LIN {X 0,Y 385.568,Z 378.768,A -85,B 0,C 180,E1 18476.822,E2 18476.822} C_VEL
LIN {X 0,Y 385.563,Z 378.767,A -85,B 0,C 180,E1 18472.892,E2 18472.892} C_VEL
LIN {X 0,Y 385.562,Z 378.769,A -85,B 0,C 180,E1 18468.915,E2 18468.915} C_VEL
LIN {X 0,Y 385.555,Z 378.77,A -85,B 0,C 180,E1 18465.03,E2 18465.03} C_VEL
LIN {X 0,Y 385.557,Z 378.769,A -85,B 0,C 180,E1 18461.064,E2 18461.064} C_VEL
LIN {X 0,Y 385.556,Z 378.767,A -85,B 0,C 180,E1 18457.001,E2 18457.001} C_VEL
LIN {X 0,Y 385.568,Z 378.766,A -85,B 0,C 180,E1 18454.536,E2 18454.536} C_VEL
LIN {X 0,Y 384.625,Z 378.889,A -85,B 0,C 180,E1 18453.392,E2 18453.392} C_VEL
LIN {X 0,Y 380.036,Z 379.462,A -85,B 0,C 180,E1 18451.232,E2 18451.232} C_VEL
LIN {X 0,Y 377.78,Z 379.738,A -85,B 0,C 180,E1 18449.743,E2 18449.743} C_VEL
LIN {X 0,Y 377.623,Z 379.753,A -85,B 0,C 180,E1 18449.318,E2 18449.318} C_VEL
LIN {X 0,Y 377.624,Z 379.757,A -85,B 0,C 180,E1 18445.292,E2 18445.292} C_VEL
LIN {X 0,Y 377.628,Z 379.756,A -85,B 0,C 180,E1 18441.32,E2 18441.32} C_VEL
LIN {X 0,Y 377.629,Z 379.756,A -85,B 0,C 180,E1 18437.305,E2 18437.305} C_VEL
LIN {X 0,Y 377.638,Z 379.756,A -85,B 0,C 180,E1 18433.384,E2 18433.384} C_VEL
LIN {X 0,Y 377.639,Z 379.756,A -85,B 0,C 180,E1 18429.382,E2 18429.382} C_VEL
LIN {X 0,Y 377.647,Z 379.757,A -85,B 0,C 180,E1 18425.438,E2 18425.438} C_VEL
LIN {X 0,Y 377.646,Z 379.757,A -85,B 0,C 180,E1 18421.366,E2 18421.366} C_VEL
LIN {X 0,Y 377.655,Z 379.76,A -85,B 0,C 180,E1 18417.489,E2 18417.489} C_VEL
LIN {X 0,Y 377.649,Z 379.762,A -85,B 0,C 180,E1 18413.343,E2 18413.343} C_VEL
LIN {X 0,Y 377.656,Z 379.759,A -85,B 0,C 180,E1 18409.36,E2 18409.36} C_VEL
LIN {X 0,Y 377.646,Z 379.758,A -85,B 0,C 180,E1 18405.23,E2 18405.23} C_VEL
LIN {X 0,Y 377.654,Z 379.759,A -85,B 0,C 180,E1 18401.242,E2 18401.242} C_VEL
LIN {X 0,Y 377.626,Z 379.853,A -85,B 0,C 180,E1 18398.318,E2 18398.318} C_VEL
LIN {X 0,Y 382.854,Z 398.245,A -85,B 0,C 180,E1 18394.648,E2 18394.648} C_VEL
LIN {X 0,Y 387.617,Z 416.474,A -85,B 0,C 180,E1 18391.231,E2 18391.231} C_VEL
LIN {X 0,Y 387.818,Z 419.084,A -85,B 0,C 180,E1 18390.79,E2 18390.79} C_VEL
LIN {X 0,Y 385.139,Z 446.418,A -85,B 0,C 180,E1 18386.578,E2 18386.578} C_VEL
LIN {X 0,Y 382.717,Z 474.798,A -85,B 0,C 180,E1 18382.261,E2 18382.261} C_VEL
LIN {X 0,Y 382.494,Z 478.618,A -85,B 0,C 180,E1 18381.736,E2 18381.736} C_VEL
LIN {X 0,Y 386.108,Z 507.081,A -85,B 0,C 180,E1 18380.765,E2 18380.765} C_VEL
LIN {X 0,Y 383,Z 605.391,A -85,B 0,C 180,E1 18378.257,E2 18378.257} C_VEL
LIN {X 0,Y 382.474,Z 621.514,A -85,B 0,C 180,E1 18377.574,E2 18377.574} C_VEL
LIN {X 0,Y 381.748,Z 637.809,A -85,B 0,C 180,E1 18376.588,E2 18376.588} C_VEL
LIN {X 0,Y 380.898,Z 652.808,A -85,B 0,C 180,E1 18375.375,E2 18375.375} C_VEL
LIN {X 0,Y 380.04,Z 667.287,A -85,B 0,C 180,E1 18373.852,E2 18373.852} C_VEL
LIN {X 0,Y 379.254,Z 679.79,A -85,B 0,C 180,E1 18372.176,E2 18372.176} C_VEL
LIN {X 0,Y 378.638,Z 689.823,A -85,B 0,C 180,E1 18370.499,E2 18370.499} C_VEL
LIN {X 0,Y 378.11,Z 699.296,A -85,B 0,C 180,E1 18368.508,E2 18368.508} C_VEL
LIN {X 0,Y 377.757,Z 706.98,A -85,B 0,C 180,E1 18366.383,E2 18366.383} C_VEL
LIN {X 0,Y 377.578,Z 712.647,A -85,B 0,C 180,E1 18364.252,E2 18364.252} C_VEL
LIN {X 0,Y 377.575,Z 716.712,A -85,B 0,C 180,E1 18361.973,E2 18361.973} C_VEL
LIN {X 0,Y 377.711,Z 718.764,A -85,B 0,C 180,E1 18359.697,E2 18359.697} C_VEL
LIN {X 0,Y 377.991,Z 718.987,A -85,B 0,C 180,E1 18357.575,E2 18357.575} C_VEL
LIN {X 0,Y 378.448,Z 717.311,A -85,B 0,C 180,E1 18355.302,E2 18355.302} C_VEL
LIN {X 0,Y 379.087,Z 713.986,A -85,B 0,C 180,E1 18353.184,E2 18353.184} C_VEL
LIN {X 0,Y 379.922,Z 708.776,A -85,B 0,C 180,E1 18351.068,E2 18351.068} C_VEL
LIN {X 0,Y 380.924,Z 702.081,A -85,B 0,C 180,E1 18349.106,E2 18349.106} C_VEL
LIN {X 0,Y 382.183,Z 693.35,A -85,B 0,C 180,E1 18347.152,E2 18347.152} C_VEL
LIN {X 0,Y 383.553,Z 682.949,A -85,B 0,C 180,E1 18345.353,E2 18345.353} C_VEL
LIN {X 0,Y 385.011,Z 671.037,A -85,B 0,C 180,E1 18343.712,E2 18343.712} C_VEL
LIN {X 0,Y 386.54,Z 657.419,A -85,B 0,C 180,E1 18342.228,E2 18342.228} C_VEL
LIN {X 0,Y 388.097,Z 641.658,A -85,B 0,C 180,E1 18340.902,E2 18340.902} C_VEL
LIN {X 0,Y 389.492,Z 625.098,A -85,B 0,C 180,E1 18339.841,E2 18339.841} C_VEL
LIN {X 0,Y 390.722,Z 606.654,A -85,B 0,C 180,E1 18339.007,E2 18339.007} C_VEL
LIN {X 0,Y 399.256,Z 512.543,A -85,B 0,C 180,E1 18335.651,E2 18335.651} C_VEL
LIN {X 0,Y 396.949,Z 494.285,A -85,B 0,C 180,E1 18334.363,E2 18334.363} C_VEL
LIN {X 0,Y 394.241,Z 477.824,A -85,B 0,C 180,E1 18332.96,E2 18332.96} C_VEL
LIN {X 0,Y 399.544,Z 456.144,A -85,B 0,C 180,E1 18328.968,E2 18328.968} C_VEL
LIN {X 0,Y 403.464,Z 443.382,A -85,B 0,C 180,E1 18326.452,E2 18326.452} C_VEL
LIN {X 0,Y 403,Z 437.068,A -85,B 0,C 180,E1 18324.16,E2 18324.16} C_VEL
LIN {X 0,Y 402.5,Z 432.282,A -85,B 0,C 180,E1 18321.72,E2 18321.72} C_VEL
LIN {X 0,Y 402.322,Z 430.143,A -85,B 0,C 180,E1 18319.934,E2 18319.934} C_VEL
LIN {X 0,Y 402.691,Z 428.705,A -85,B 0,C 180,E1 18317.304,E2 18317.304} C_VEL
LIN {X 0,Y 402.969,Z 429.281,A -85,B 0,C 180,E1 18315.814,E2 18315.814} C_VEL
LIN {X 0,Y 403.921,Z 432.089,A -85,B 0,C 180,E1 18313.29,E2 18313.29} C_VEL
LIN {X 0,Y 405.118,Z 436.513,A -85,B 0,C 180,E1 18311.17,E2 18311.17} C_VEL
LIN {X 0,Y 406.456,Z 442.396,A -85,B 0,C 180,E1 18309.206,E2 18309.206} C_VEL
LIN {X 0,Y 406.774,Z 444.189,A -85,B 0,C 180,E1 18308.724,E2 18308.724} C_VEL
LIN {X 0,Y 400.249,Z 465.939,A -85,B 0,C 180,E1 18305.772,E2 18305.772} C_VEL
LIN {X 0,Y 399.345,Z 470.309,A -85,B 0,C 180,E1 18305.241,E2 18305.241} C_VEL
LIN {X 0,Y 400.489,Z 482.433,A -85,B 0,C 180,E1 18304.586,E2 18304.586} C_VEL
LIN {X 0,Y 400.887,Z 494.633,A -85,B 0,C 180,E1 18304.069,E2 18304.069} C_VEL
LIN {X 0,Y 395.517,Z 583.729,A -85,B 0,C 180,E1 18301.729,E2 18301.729} C_VEL
LIN {X 0,Y 392.122,Z 659.98,A -85,B 0,C 180,E1 18299.871,E2 18299.871} C_VEL
LIN {X 0,Y 390.555,Z 679.348,A -85,B 0,C 180,E1 18299.137,E2 18299.137} C_VEL
LIN {X 0,Y 388.108,Z 704.589,A -85,B 0,C 180,E1 18297.795,E2 18297.795} C_VEL
LIN {X 0,Y 386.353,Z 722.572,A -85,B 0,C 180,E1 18296.597,E2 18296.597} C_VEL
LIN {X 0,Y 384.511,Z 739.688,A -85,B 0,C 180,E1 18295.161,E2 18295.161} C_VEL
LIN {X 0,Y 382.682,Z 755.778,A -85,B 0,C 180,E1 18293.497,E2 18293.497} C_VEL
LIN {X 0,Y 380.908,Z 771.145,A -85,B 0,C 180,E1 18291.561,E2 18291.561} C_VEL
LIN {X 0,Y 379.335,Z 785.195,A -85,B 0,C 180,E1 18289.397,E2 18289.397} C_VEL
LIN {X 0,Y 378.118,Z 796.867,A -85,B 0,C 180,E1 18287.227,E2 18287.227} C_VEL
LIN {X 0,Y 377.209,Z 807.217,A -85,B 0,C 180,E1 18284.899,E2 18284.899} C_VEL
LIN {X 0,Y 376.589,Z 816.167,A -85,B 0,C 180,E1 18282.419,E2 18282.419} C_VEL
LIN {X 0,Y 376.257,Z 823.621,A -85,B 0,C 180,E1 18279.792,E2 18279.792} C_VEL
LIN {X 0,Y 376.195,Z 829.193,A -85,B 0,C 180,E1 18277.176,E2 18277.176} C_VEL
LIN {X 0,Y 376.215,Z 833.01,A -85,B 0,C 180,E1 18274.573,E2 18274.573} C_VEL
LIN {X 0,Y 376.278,Z 835.161,A -85,B 0,C 180,E1 18271.98,E2 18271.98} C_VEL
LIN {X 0,Y 376.295,Z 835.689,A -85,B 0,C 180,E1 18269.391,E2 18269.391} C_VEL
LIN {X 0,Y 376.236,Z 834.596,A -85,B 0,C 180,E1 18266.801,E2 18266.801} C_VEL
LIN {X 0,Y 376.173,Z 831.658,A -85,B 0,C 180,E1 18264.05,E2 18264.05} C_VEL
LIN {X 0,Y 376.187,Z 827.071,A -85,B 0,C 180,E1 18261.389,E2 18261.389} C_VEL
LIN {X 0,Y 376.416,Z 820.496,A -85,B 0,C 180,E1 18258.664,E2 18258.664} C_VEL
LIN {X 0,Y 376.976,Z 812.236,A -85,B 0,C 180,E1 18256.033,E2 18256.033} C_VEL
LIN {X 0,Y 377.868,Z 802.515,A -85,B 0,C 180,E1 18253.553,E2 18253.553} C_VEL
LIN {X 0,Y 379.228,Z 790.6,A -85,B 0,C 180,E1 18251.077,E2 18251.077} C_VEL
LIN {X 0,Y 380.955,Z 777.066,A -85,B 0,C 180,E1 18248.765,E2 18248.765} C_VEL
LIN {X 0,Y 382.953,Z 762.46,A -85,B 0,C 180,E1 18246.699,E2 18246.699} C_VEL
LIN {X 0,Y 385.216,Z 746.307,A -85,B 0,C 180,E1 18244.806,E2 18244.806} C_VEL
LIN {X 0,Y 387.585,Z 729.237,A -85,B 0,C 180,E1 18243.163,E2 18243.163} C_VEL
LIN {X 0,Y 389.976,Z 711.341,A -85,B 0,C 180,E1 18241.768,E2 18241.768} C_VEL
LIN {X 0,Y 392.36,Z 692.082,A -85,B 0,C 180,E1 18240.581,E2 18240.581} C_VEL
LIN {X 0,Y 394.622,Z 671.766,A -85,B 0,C 180,E1 18239.633,E2 18239.633} C_VEL
LIN {X 0,Y 396.506,Z 650.21,A -85,B 0,C 180,E1 18238.909,E2 18238.909} C_VEL
LIN {X 0,Y 402.188,Z 575.648,A -85,B 0,C 180,E1 18236.758,E2 18236.758} C_VEL
LIN {X 0,Y 410.35,Z 494.898,A -85,B 0,C 180,E1 18234.274,E2 18234.274} C_VEL
LIN {X 0,Y 410.677,Z 466.837,A -85,B 0,C 180,E1 18232.704,E2 18232.704} C_VEL
LIN {X 0,Y 411.103,Z 441.518,A -85,B 0,C 180,E1 18231.022,E2 18231.022} C_VEL
LIN {X 0,Y 409.658,Z 433.244,A -85,B 0,C 180,E1 18229.7,E2 18229.7} C_VEL
LIN {X 0,Y 409.278,Z 423.175,A -85,B 0,C 180,E1 18227.75,E2 18227.75} C_VEL
LIN {X 0,Y 409.104,Z 422.172,A -85,B 0,C 180,E1 18227.391,E2 18227.391} C_VEL
LIN {X 0,Y 408.012,Z 420.874,A -85,B 0,C 180,E1 18225.689,E2 18225.689} C_VEL
LIN {X 0,Y 407.37,Z 421.427,A -85,B 0,C 180,E1 18223.8,E2 18223.8} C_VEL
LIN {X 0,Y 407.668,Z 422.762,A -85,B 0,C 180,E1 18222.318,E2 18222.318} C_VEL
LIN {X 0,Y 408.394,Z 426.503,A -85,B 0,C 180,E1 18220.484,E2 18220.484} C_VEL
LIN {X 0,Y 410.334,Z 430.82,A -85,B 0,C 180,E1 18219.131,E2 18219.131} C_VEL
LIN {X 0,Y 413.028,Z 437.043,A -85,B 0,C 180,E1 18217.692,E2 18217.692} C_VEL
LIN {X 0,Y 415.906,Z 444.855,A -85,B 0,C 180,E1 18216.395,E2 18216.395} C_VEL
LIN {X 0,Y 406.008,Z 529.242,A -85,B 0,C 180,E1 18213.781,E2 18213.781} C_VEL
LIN {X 0,Y 399.705,Z 599.781,A -85,B 0,C 180,E1 18211.689,E2 18211.689} C_VEL
LIN {X 0,Y 397.377,Z 632.042,A -85,B 0,C 180,E1 18210.705,E2 18210.705} C_VEL
LIN {X 0,Y 395.669,Z 651.221,A -85,B 0,C 180,E1 18209.856,E2 18209.856} C_VEL
LIN {X 0,Y 393.692,Z 669.727,A -85,B 0,C 180,E1 18208.768,E2 18208.768} C_VEL
LIN {X 0,Y 391.499,Z 687.412,A -85,B 0,C 180,E1 18207.45,E2 18207.45} C_VEL
LIN {X 0,Y 389.183,Z 704.226,A -85,B 0,C 180,E1 18205.897,E2 18205.897} C_VEL
LIN {X 0,Y 386.804,Z 719.968,A -85,B 0,C 180,E1 18204.105,E2 18204.105} C_VEL
LIN {X 0,Y 384.547,Z 734.138,A -85,B 0,C 180,E1 18202.149,E2 18202.149} C_VEL
LIN {X 0,Y 382.475,Z 746.857,A -85,B 0,C 180,E1 18200.026,E2 18200.026} C_VEL
LIN {X 0,Y 380.653,Z 758.153,A -85,B 0,C 180,E1 18197.74,E2 18197.74} C_VEL
LIN {X 0,Y 379.124,Z 768.019,A -85,B 0,C 180,E1 18195.291,E2 18195.291} C_VEL
LIN {X 0,Y 377.928,Z 776.403,A -85,B 0,C 180,E1 18192.685,E2 18192.685} C_VEL
LIN {X 0,Y 377.112,Z 782.884,A -85,B 0,C 180,E1 18190.078,E2 18190.078} C_VEL
LIN {X 0,Y 376.581,Z 787.886,A -85,B 0,C 180,E1 18187.322,E2 18187.322} C_VEL
LIN {X 0,Y 376.294,Z 791.101,A -85,B 0,C 180,E1 18184.572,E2 18184.572} C_VEL
LIN {X 0,Y 376.172,Z 792.605,A -85,B 0,C 180,E1 18181.828,E2 18181.828} C_VEL
LIN {X 0,Y 376.132,Z 792.422,A -85,B 0,C 180,E1 18179.086,E2 18179.086} C_VEL
LIN {X 0,Y 376.15,Z 790.549,A -85,B 0,C 180,E1 18176.342,E2 18176.342} C_VEL
LIN {X 0,Y 376.279,Z 786.94,A -85,B 0,C 180,E1 18173.592,E2 18173.592} C_VEL
LIN {X 0,Y 376.558,Z 781.862,A -85,B 0,C 180,E1 18170.987,E2 18170.987} C_VEL
LIN {X 0,Y 377.072,Z 775.014,A -85,B 0,C 180,E1 18168.374,E2 18168.374} C_VEL
LIN {X 0,Y 377.837,Z 766.791,A -85,B 0,C 180,E1 18165.909,E2 18165.909} C_VEL
LIN {X 0,Y 378.931,Z 756.558,A -85,B 0,C 180,E1 18163.443,E2 18163.443} C_VEL
LIN {X 0,Y 380.298,Z 744.838,A -85,B 0,C 180,E1 18161.132,E2 18161.132} C_VEL
LIN {X 0,Y 381.966,Z 731.098,A -85,B 0,C 180,E1 18158.904,E2 18158.904} C_VEL
LIN {X 0,Y 383.693,Z 716.811,A -85,B 0,C 180,E1 18156.99,E2 18156.99} C_VEL
LIN {X 0,Y 385.533,Z 700.907,A -85,B 0,C 180,E1 18155.23,E2 18155.23} C_VEL
LIN {X 0,Y 387.318,Z 684.321,A -85,B 0,C 180,E1 18153.73,E2 18153.73} C_VEL
LIN {X 0,Y 389.016,Z 666.608,A -85,B 0,C 180,E1 18152.442,E2 18152.442} C_VEL
LIN {X 0,Y 390.489,Z 647.986,A -85,B 0,C 180,E1 18151.391,E2 18151.391} C_VEL
LIN {X 0,Y 391.72,Z 628.44,A -85,B 0,C 180,E1 18150.581,E2 18150.581} C_VEL
LIN {X 0,Y 392.684,Z 605.735,A -85,B 0,C 180,E1 18149.961,E2 18149.961} C_VEL
LIN {X 0,Y 399.153,Z 438.469,A -85,B 0,C 180,E1 18146.166,E2 18146.166} C_VEL
LIN {X 0,Y 397.46,Z 429.615,A -85,B 0,C 180,E1 18145.793,E2 18145.793} C_VEL
LIN {X 0,Y 388.641,Z 410.821,A -85,B 0,C 180,E1 18144.515,E2 18144.515} C_VEL
LIN {X 0,Y 381.033,Z 389.206,A -85,B 0,C 180,E1 18141.322,E2 18141.322} C_VEL
LIN {X 0,Y 377.626,Z 379.756,A -85,B 0,C 180,E1 18139.855,E2 18139.855} C_VEL
LIN {X 0,Y 377.631,Z 379.759,A -85,B 0,C 180,E1 18135.865,E2 18135.865} C_VEL
LIN {X 0,Y 377.632,Z 379.757,A -85,B 0,C 180,E1 18131.853,E2 18131.853} C_VEL
LIN {X 0,Y 377.635,Z 379.759,A -85,B 0,C 180,E1 18127.899,E2 18127.899} C_VEL
LIN {X 0,Y 377.642,Z 379.759,A -85,B 0,C 180,E1 18123.963,E2 18123.963} C_VEL
LIN {X 0,Y 377.651,Z 379.756,A -85,B 0,C 180,E1 18120.026,E2 18120.026} C_VEL
LIN {X 0,Y 377.654,Z 379.757,A -85,B 0,C 180,E1 18116.072,E2 18116.072} C_VEL
LIN {X 0,Y 377.664,Z 379.756,A -85,B 0,C 180,E1 18112.083,E2 18112.083} C_VEL
LIN {X 0,Y 377.657,Z 379.755,A -85,B 0,C 180,E1 18108.045,E2 18108.045} C_VEL
LIN {X 0,Y 377.657,Z 379.753,A -85,B 0,C 180,E1 18103.941,E2 18103.941} C_VEL
LIN {X 0,Y 377.654,Z 379.755,A -85,B 0,C 180,E1 18099.909,E2 18099.909} C_VEL
LIN {X 0,Y 377.66,Z 379.756,A -85,B 0,C 180,E1 18095.927,E2 18095.927} C_VEL
LIN {X 0,Y 377.653,Z 379.757,A -85,B 0,C 180,E1 18091.821,E2 18091.821} C_VEL
LIN {X 0,Y 377.623,Z 379.753,A -85,B 0,C 180,E1 18089.318,E2 18089.318} C_VEL
LIN {X 0,Y 376.599,Z 379.881,A -85,B 0,C 180,E1 18088.149,E2 18088.149} C_VEL
LIN {X 0,Y 370.113,Z 380.695,A -85,B 0,C 180,E1 18084.764,E2 18084.764} C_VEL
LIN {X 0,Y 369.72,Z 380.745,A -85,B 0,C 180,E1 18083.987,E2 18083.987} C_VEL
LIN {X 0,Y 369.717,Z 380.747,A -85,B 0,C 180,E1 18079.867,E2 18079.867} C_VEL
LIN {X 0,Y 369.728,Z 380.746,A -85,B 0,C 180,E1 18075.753,E2 18075.753} C_VEL
LIN {X 0,Y 369.712,Z 380.749,A -85,B 0,C 180,E1 18071.553,E2 18071.553} C_VEL
LIN {X 0,Y 369.707,Z 380.746,A -85,B 0,C 180,E1 18067.416,E2 18067.416} C_VEL
LIN {X 0,Y 369.703,Z 380.745,A -85,B 0,C 180,E1 18063.324,E2 18063.324} C_VEL
LIN {X 0,Y 369.704,Z 380.749,A -85,B 0,C 180,E1 18059.32,E2 18059.32} C_VEL
LIN {X 0,Y 369.698,Z 380.752,A -85,B 0,C 180,E1 18055.204,E2 18055.204} C_VEL
LIN {X 0,Y 369.697,Z 380.751,A -85,B 0,C 180,E1 18051.137,E2 18051.137} C_VEL
LIN {X 0,Y 369.699,Z 380.747,A -85,B 0,C 180,E1 18047.133,E2 18047.133} C_VEL
LIN {X 0,Y 369.7,Z 380.748,A -85,B 0,C 180,E1 18043.095,E2 18043.095} C_VEL
LIN {X 0,Y 369.698,Z 380.75,A -85,B 0,C 180,E1 18039.062,E2 18039.062} C_VEL
LIN {X 0,Y 369.757,Z 381.22,A -85,B 0,C 180,E1 18038.855,E2 18038.855} C_VEL
LIN {X 0,Y 374.774,Z 398.754,A -85,B 0,C 180,E1 18035.276,E2 18035.276} C_VEL
LIN {X 0,Y 379.528,Z 416.859,A -85,B 0,C 180,E1 18031.796,E2 18031.796} C_VEL
LIN {X 0,Y 380.268,Z 420.648,A -85,B 0,C 180,E1 18031.109,E2 18031.109} C_VEL
LIN {X 0,Y 377.525,Z 447.325,A -85,B 0,C 180,E1 18026.929,E2 18026.929} C_VEL
LIN {X 0,Y 375.004,Z 475.468,A -85,B 0,C 180,E1 18022.578,E2 18022.578} C_VEL
LIN {X 0,Y 374.832,Z 478.495,A -85,B 0,C 180,E1 18022.165,E2 18022.165} C_VEL
LIN {X 0,Y 378.508,Z 508.02,A -85,B 0,C 180,E1 18021.131,E2 18021.131} C_VEL
LIN {X 0,Y 375.259,Z 606.055,A -85,B 0,C 180,E1 18018.551,E2 18018.551} C_VEL
LIN {X 0,Y 374.724,Z 621.863,A -85,B 0,C 180,E1 18017.87,E2 18017.87} C_VEL
LIN {X 0,Y 373.964,Z 638.363,A -85,B 0,C 180,E1 18016.856,E2 18016.856} C_VEL
LIN {X 0,Y 373.037,Z 654.174,A -85,B 0,C 180,E1 18015.547,E2 18015.547} C_VEL
LIN {X 0,Y 372.156,Z 668.567,A -85,B 0,C 180,E1 18013.993,E2 18013.993} C_VEL
LIN {X 0,Y 371.305,Z 681.716,A -85,B 0,C 180,E1 18012.176,E2 18012.176} C_VEL
LIN {X 0,Y 370.611,Z 692.62,A -85,B 0,C 180,E1 18010.257,E2 18010.257} C_VEL
LIN {X 0,Y 370.14,Z 701.073,A -85,B 0,C 180,E1 18008.388,E2 18008.388} C_VEL
LIN {X 0,Y 369.798,Z 708.702,A -85,B 0,C 180,E1 18006.209,E2 18006.209} C_VEL
LIN {X 0,Y 369.639,Z 714.231,A -85,B 0,C 180,E1 18004.033,E2 18004.033} C_VEL
LIN {X 0,Y 369.657,Z 717.995,A -85,B 0,C 180,E1 18001.86,E2 18001.86} C_VEL
LIN {X 0,Y 369.826,Z 720.072,A -85,B 0,C 180,E1 17999.535,E2 17999.535} C_VEL
LIN {X 0,Y 370.141,Z 720.31,A -85,B 0,C 180,E1 17997.368,E2 17997.368} C_VEL
LIN {X 0,Y 370.665,Z 718.662,A -85,B 0,C 180,E1 17995.048,E2 17995.048} C_VEL
LIN {X 0,Y 371.371,Z 715.331,A -85,B 0,C 180,E1 17992.886,E2 17992.886} C_VEL
LIN {X 0,Y 372.384,Z 709.742,A -85,B 0,C 180,E1 17990.573,E2 17990.573} C_VEL
LIN {X 0,Y 373.51,Z 702.92,A -85,B 0,C 180,E1 17988.575,E2 17988.575} C_VEL
LIN {X 0,Y 374.897,Z 694.028,A -85,B 0,C 180,E1 17986.583,E2 17986.583} C_VEL
LIN {X 0,Y 376.424,Z 683.581,A -85,B 0,C 180,E1 17984.754,E2 17984.754} C_VEL
LIN {X 0,Y 378.006,Z 671.493,A -85,B 0,C 180,E1 17983.085,E2 17983.085} C_VEL
LIN {X 0,Y 379.69,Z 657.785,A -85,B 0,C 180,E1 17981.579,E2 17981.579} C_VEL
LIN {X 0,Y 381.356,Z 642.408,A -85,B 0,C 180,E1 17980.263,E2 17980.263} C_VEL
LIN {X 0,Y 382.845,Z 626.056,A -85,B 0,C 180,E1 17979.195,E2 17979.195} C_VEL
LIN {X 0,Y 384.223,Z 607.725,A -85,B 0,C 180,E1 17978.334,E2 17978.334} C_VEL
LIN {X 0,Y 393.311,Z 516.535,A -85,B 0,C 180,E1 17974.994,E2 17974.994} C_VEL
LIN {X 0,Y 393.265,Z 512.705,A -85,B 0,C 180,E1 17974.781,E2 17974.781} C_VEL
LIN {X 0,Y 391.072,Z 494.356,A -85,B 0,C 180,E1 17973.391,E2 17973.391} C_VEL
LIN {X 0,Y 388.486,Z 477.673,A -85,B 0,C 180,E1 17971.86,E2 17971.86} C_VEL
LIN {X 0,Y 394.363,Z 456.593,A -85,B 0,C 180,E1 17967.83,E2 17967.83} C_VEL
LIN {X 0,Y 397.392,Z 447.84,A -85,B 0,C 180,E1 17966.044,E2 17966.044} C_VEL
LIN {X 0,Y 397.108,Z 441.732,A -85,B 0,C 180,E1 17963.68,E2 17963.68} C_VEL
LIN {X 0,Y 396.836,Z 437.574,A -85,B 0,C 180,E1 17961.329,E2 17961.329} C_VEL
LIN {X 0,Y 396.752,Z 435.698,A -85,B 0,C 180,E1 17959.559,E2 17959.559} C_VEL
LIN {X 0,Y 397.374,Z 434.596,A -85,B 0,C 180,E1 17957.009,E2 17957.009} C_VEL
LIN {X 0,Y 397.644,Z 435.792,A -85,B 0,C 180,E1 17955.16,E2 17955.16} C_VEL
LIN {X 0,Y 398.498,Z 438.429,A -85,B 0,C 180,E1 17953.102,E2 17953.102} C_VEL
LIN {X 0,Y 399.604,Z 442.486,A -85,B 0,C 180,E1 17951.152,E2 17951.152} C_VEL
LIN {X 0,Y 400.71,Z 448.361,A -85,B 0,C 180,E1 17949.238,E2 17949.238} C_VEL
LIN {X 0,Y 393.838,Z 469.66,A -85,B 0,C 180,E1 17946.266,E2 17946.266} C_VEL
LIN {X 0,Y 394.183,Z 474.345,A -85,B 0,C 180,E1 17945.929,E2 17945.929} C_VEL
LIN {X 0,Y 394.979,Z 485.606,A -85,B 0,C 180,E1 17945.307,E2 17945.307} C_VEL
LIN {X 0,Y 395.146,Z 496.037,A -85,B 0,C 180,E1 17944.853,E2 17944.853} C_VEL
LIN {X 0,Y 389.298,Z 582.532,A -85,B 0,C 180,E1 17942.487,E2 17942.487} C_VEL
LIN {X 0,Y 385.449,Z 659.08,A -85,B 0,C 180,E1 17940.54,E2 17940.54} C_VEL
LIN {X 0,Y 383.743,Z 678.68,A -85,B 0,C 180,E1 17939.776,E2 17939.776} C_VEL
LIN {X 0,Y 381.764,Z 696.563,A -85,B 0,C 180,E1 17938.81,E2 17938.81} C_VEL
LIN {X 0,Y 378.36,Z 726.053,A -85,B 0,C 180,E1 17936.695,E2 17936.695} C_VEL
LIN {X 0,Y 376.412,Z 743.188,A -85,B 0,C 180,E1 17935.151,E2 17935.151} C_VEL
LIN {X 0,Y 374.482,Z 759.339,A -85,B 0,C 180,E1 17933.359,E2 17933.359} C_VEL
LIN {X 0,Y 372.648,Z 774.627,A -85,B 0,C 180,E1 17931.288,E2 17931.288} C_VEL
LIN {X 0,Y 371.176,Z 787.441,A -85,B 0,C 180,E1 17929.186,E2 17929.186} C_VEL
LIN {X 0,Y 369.909,Z 799.423,A -85,B 0,C 180,E1 17926.811,E2 17926.811} C_VEL
LIN {X 0,Y 369.015,Z 809.859,A -85,B 0,C 180,E1 17924.275,E2 17924.275} C_VEL
LIN {X 0,Y 368.466,Z 818.204,A -85,B 0,C 180,E1 17921.743,E2 17921.743} C_VEL
LIN {X 0,Y 368.221,Z 825.095,A -85,B 0,C 180,E1 17919.061,E2 17919.061} C_VEL
LIN {X 0,Y 368.194,Z 830.219,A -85,B 0,C 180,E1 17916.332,E2 17916.332} C_VEL
LIN {X 0,Y 368.25,Z 833.553,A -85,B 0,C 180,E1 17913.58,E2 17913.58} C_VEL
LIN {X 0,Y 368.314,Z 835.072,A -85,B 0,C 180,E1 17910.933,E2 17910.933} C_VEL
LIN {X 0,Y 368.289,Z 834.952,A -85,B 0,C 180,E1 17908.289,E2 17908.289} C_VEL
LIN {X 0,Y 368.213,Z 833.212,A -85,B 0,C 180,E1 17905.639,E2 17905.639} C_VEL
LIN {X 0,Y 368.173,Z 829.84,A -85,B 0,C 180,E1 17902.98,E2 17902.98} C_VEL
LIN {X 0,Y 368.25,Z 824.693,A -85,B 0,C 180,E1 17900.266,E2 17900.266} C_VEL
LIN {X 0,Y 368.633,Z 817.487,A -85,B 0,C 180,E1 17897.468,E2 17897.468} C_VEL
LIN {X 0,Y 369.389,Z 808.577,A -85,B 0,C 180,E1 17894.778,E2 17894.778} C_VEL
LIN {X 0,Y 370.55,Z 798.165,A -85,B 0,C 180,E1 17892.247,E2 17892.247} C_VEL
LIN {X 0,Y 372.099,Z 786.335,A -85,B 0,C 180,E1 17889.882,E2 17889.882} C_VEL
LIN {X 0,Y 374.141,Z 772.067,A -85,B 0,C 180,E1 17887.533,E2 17887.533} C_VEL
LIN {X 0,Y 376.469,Z 756.598,A -85,B 0,C 180,E1 17885.434,E2 17885.434} C_VEL
LIN {X 0,Y 379.063,Z 739.494,A -85,B 0,C 180,E1 17883.527,E2 17883.527} C_VEL
LIN {X 0,Y 381.648,Z 722.172,A -85,B 0,C 180,E1 17881.949,E2 17881.949} C_VEL
LIN {X 0,Y 384.372,Z 703.127,A -85,B 0,C 180,E1 17880.551,E2 17880.551} C_VEL
LIN {X 0,Y 386.91,Z 683.606,A -85,B 0,C 180,E1 17879.44,E2 17879.44} C_VEL
LIN {X 0,Y 389.28,Z 662.827,A -85,B 0,C 180,E1 17878.563,E2 17878.563} C_VEL
LIN {X 0,Y 397.731,Z 566.301,A -85,B 0,C 180,E1 17875.614,E2 17875.614} C_VEL
LIN {X 0,Y 405.715,Z 495.632,A -85,B 0,C 180,E1 17873.344,E2 17873.344} C_VEL
LIN {X 0,Y 406.584,Z 468.128,A -85,B 0,C 180,E1 17871.727,E2 17871.727} C_VEL
LIN {X 0,Y 407.556,Z 445.658,A -85,B 0,C 180,E1 17870.185,E2 17870.185} C_VEL
LIN {X 0,Y 405.976,Z 433.544,A -85,B 0,C 180,E1 17868.054,E2 17868.054} C_VEL
LIN {X 0,Y 406.086,Z 429.468,A -85,B 0,C 180,E1 17867.19,E2 17867.19} C_VEL
LIN {X 0,Y 404.946,Z 428.278,A -85,B 0,C 180,E1 17865.474,E2 17865.474} C_VEL
LIN {X 0,Y 404.285,Z 429.145,A -85,B 0,C 180,E1 17863.355,E2 17863.355} C_VEL
LIN {X 0,Y 404.63,Z 430.151,A -85,B 0,C 180,E1 17862.475,E2 17862.475} C_VEL
LIN {X 0,Y 405.92,Z 433.782,A -85,B 0,C 180,E1 17860.799,E2 17860.799} C_VEL
LIN {X 0,Y 407.996,Z 438.744,A -85,B 0,C 180,E1 17859.248,E2 17859.248} C_VEL
LIN {X 0,Y 410.653,Z 445.868,A -85,B 0,C 180,E1 17857.72,E2 17857.72} C_VEL
LIN {X 0,Y 411.508,Z 448.898,A -85,B 0,C 180,E1 17857.25,E2 17857.25} C_VEL
LIN {X 0,Y 400.841,Z 531.541,A -85,B 0,C 180,E1 17854.613,E2 17854.613} C_VEL
LIN {X 0,Y 393.943,Z 600.579,A -85,B 0,C 180,E1 17852.482,E2 17852.482} C_VEL
LIN {X 0,Y 391.321,Z 632.966,A -85,B 0,C 180,E1 17851.453,E2 17851.453} C_VEL
LIN {X 0,Y 389.396,Z 652.461,A -85,B 0,C 180,E1 17850.558,E2 17850.558} C_VEL
LIN {X 0,Y 387.138,Z 671.673,A -85,B 0,C 180,E1 17849.387,E2 17849.387} C_VEL
LIN {X 0,Y 384.622,Z 690.196,A -85,B 0,C 180,E1 17847.947,E2 17847.947} C_VEL
LIN {X 0,Y 381.965,Z 707.5,A -85,B 0,C 180,E1 17846.256,E2 17846.256} C_VEL
LIN {X 0,Y 379.363,Z 723.309,A -85,B 0,C 180,E1 17844.359,E2 17844.359} C_VEL
LIN {X 0,Y 376.916,Z 737.466,A -85,B 0,C 180,E1 17842.293,E2 17842.293} C_VEL
LIN {X 0,Y 374.701,Z 750.038,A -85,B 0,C 180,E1 17840.067,E2 17840.067} C_VEL
LIN {X 0,Y 372.744,Z 761.258,A -85,B 0,C 180,E1 17837.645,E2 17837.645} C_VEL
LIN {X 0,Y 371.172,Z 770.617,A -85,B 0,C 180,E1 17835.147,E2 17835.147} C_VEL
LIN {X 0,Y 369.944,Z 778.528,A -85,B 0,C 180,E1 17832.487,E2 17832.487} C_VEL
LIN {X 0,Y 369.111,Z 784.607,A -85,B 0,C 180,E1 17829.826,E2 17829.826} C_VEL
LIN {X 0,Y 368.576,Z 789.202,A -85,B 0,C 180,E1 17827.012,E2 17827.012} C_VEL
LIN {X 0,Y 368.296,Z 792.037,A -85,B 0,C 180,E1 17824.203,E2 17824.203} C_VEL
LIN {X 0,Y 368.176,Z 793.176,A -85,B 0,C 180,E1 17821.4,E2 17821.4} C_VEL
LIN {X 0,Y 368.135,Z 792.623,A -85,B 0,C 180,E1 17818.599,E2 17818.599} C_VEL
LIN {X 0,Y 368.174,Z 790.372,A -85,B 0,C 180,E1 17815.795,E2 17815.795} C_VEL
LIN {X 0,Y 368.341,Z 786.367,A -85,B 0,C 180,E1 17812.983,E2 17812.983} C_VEL
LIN {X 0,Y 368.711,Z 780.503,A -85,B 0,C 180,E1 17810.163,E2 17810.163} C_VEL
LIN {X 0,Y 369.331,Z 773.099,A -85,B 0,C 180,E1 17807.492,E2 17807.492} C_VEL
LIN {X 0,Y 370.225,Z 764.263,A -85,B 0,C 180,E1 17804.973,E2 17804.973} C_VEL
LIN {X 0,Y 371.48,Z 753.349,A -85,B 0,C 180,E1 17802.455,E2 17802.455} C_VEL
LIN {X 0,Y 373.025,Z 740.812,A -85,B 0,C 180,E1 17800.098,E2 17800.098} C_VEL
LIN {X 0,Y 374.743,Z 727.156,A -85,B 0,C 180,E1 17797.983,E2 17797.983} C_VEL
LIN {X 0,Y 376.633,Z 711.922,A -85,B 0,C 180,E1 17796.035,E2 17796.035} C_VEL
LIN {X 0,Y 378.635,Z 694.806,A -85,B 0,C 180,E1 17794.245,E2 17794.245} C_VEL
LIN {X 0,Y 380.475,Z 677.603,A -85,B 0,C 180,E1 17792.789,E2 17792.789} C_VEL
LIN {X 0,Y 382.166,Z 659.406,A -85,B 0,C 180,E1 17791.564,E2 17791.564} C_VEL
LIN {X 0,Y 383.633,Z 640.009,A -85,B 0,C 180,E1 17790.575,E2 17790.575} C_VEL
LIN {X 0,Y 384.748,Z 620.348,A -85,B 0,C 180,E1 17789.864,E2 17789.864} C_VEL
LIN {X 0,Y 392.121,Z 439.692,A -85,B 0,C 180,E1 17785.626,E2 17785.626} C_VEL
LIN {X 0,Y 390.737,Z 432.763,A -85,B 0,C 180,E1 17785.323,E2 17785.323} C_VEL
LIN {X 0,Y 380.492,Z 411.017,A -85,B 0,C 180,E1 17783.779,E2 17783.779} C_VEL
LIN {X 0,Y 372.849,Z 389.506,A -85,B 0,C 180,E1 17780.538,E2 17780.538} C_VEL
LIN {X 0,Y 369.687,Z 380.75,A -85,B 0,C 180,E1 17779.173,E2 17779.173} C_VEL
LIN {X 0,Y 369.689,Z 380.749,A -85,B 0,C 180,E1 17775.097,E2 17775.097} C_VEL
LIN {X 0,Y 369.69,Z 380.746,A -85,B 0,C 180,E1 17771.011,E2 17771.011} C_VEL
LIN {X 0,Y 369.686,Z 380.748,A -85,B 0,C 180,E1 17767.073,E2 17767.073} C_VEL
LIN {X 0,Y 369.685,Z 380.749,A -85,B 0,C 180,E1 17763.024,E2 17763.024} C_VEL
LIN {X 0,Y 369.681,Z 380.745,A -85,B 0,C 180,E1 17759.119,E2 17759.119} C_VEL
LIN {X 0,Y 369.684,Z 380.746,A -85,B 0,C 180,E1 17755.034,E2 17755.034} C_VEL
LIN {X 0,Y 369.681,Z 380.744,A -85,B 0,C 180,E1 17751.075,E2 17751.075} C_VEL
LIN {X 0,Y 369.682,Z 380.742,A -85,B 0,C 180,E1 17746.984,E2 17746.984} C_VEL
LIN {X 0,Y 369.679,Z 380.742,A -85,B 0,C 180,E1 17742.973,E2 17742.973} C_VEL
LIN {X 0,Y 369.68,Z 380.742,A -85,B 0,C 180,E1 17738.868,E2 17738.868} C_VEL
LIN {X 0,Y 369.681,Z 380.744,A -85,B 0,C 180,E1 17734.81,E2 17734.81} C_VEL
LIN {X 0,Y 369.679,Z 380.746,A -85,B 0,C 180,E1 17730.775,E2 17730.775} C_VEL
LIN {X 0,Y 369.679,Z 380.742,A -85,B 0,C 180,E1 17726.744,E2 17726.744} C_VEL
LIN {X 0,Y 369.72,Z 380.745,A -85,B 0,C 180,E1 17723.987,E2 17723.987} C_VEL
LIN {X 0,Y 368.892,Z 380.848,A -85,B 0,C 180,E1 17722.877,E2 17722.877} C_VEL
LIN {X 0,Y 365.016,Z 381.328,A -85,B 0,C 180,E1 17720.961,E2 17720.961} C_VEL
LIN {X 0,Y 362.081,Z 381.694,A -85,B 0,C 180,E1 17719.25,E2 17719.25} C_VEL
LIN {X 0,Y 361.744,Z 381.735,A -85,B 0,C 180,E1 17718.543,E2 17718.543} C_VEL
LIN {X 0,Y 361.739,Z 381.737,A -85,B 0,C 180,E1 17714.612,E2 17714.612} C_VEL
LIN {X 0,Y 361.745,Z 381.737,A -85,B 0,C 180,E1 17710.48,E2 17710.48} C_VEL
LIN {X 0,Y 361.74,Z 381.735,A -85,B 0,C 180,E1 17706.545,E2 17706.545} C_VEL
LIN {X 0,Y 361.742,Z 381.735,A -85,B 0,C 180,E1 17702.51,E2 17702.51} C_VEL
LIN {X 0,Y 361.741,Z 381.738,A -85,B 0,C 180,E1 17698.506,E2 17698.506} C_VEL
LIN {X 0,Y 361.742,Z 381.741,A -85,B 0,C 180,E1 17694.323,E2 17694.323} C_VEL
LIN {X 0,Y 361.744,Z 381.739,A -85,B 0,C 180,E1 17690.21,E2 17690.21} C_VEL
LIN {X 0,Y 361.743,Z 381.737,A -85,B 0,C 180,E1 17686.171,E2 17686.171} C_VEL
LIN {X 0,Y 361.742,Z 381.739,A -85,B 0,C 180,E1 17682.195,E2 17682.195} C_VEL
LIN {X 0,Y 361.795,Z 381.852,A -85,B 0,C 180,E1 17679.552,E2 17679.552} C_VEL
LIN {X 0,Y 367.108,Z 400.55,A -85,B 0,C 180,E1 17675.652,E2 17675.652} C_VEL
LIN {X 0,Y 372.002,Z 419.365,A -85,B 0,C 180,E1 17671.971,E2 17671.971} C_VEL
LIN {X 0,Y 372.665,Z 422.619,A -85,B 0,C 180,E1 17671.366,E2 17671.366} C_VEL
LIN {X 0,Y 369.737,Z 449.932,A -85,B 0,C 180,E1 17667.021,E2 17667.021} C_VEL
LIN {X 0,Y 367.152,Z 478.102,A -85,B 0,C 180,E1 17662.614,E2 17662.614} C_VEL
LIN {X 0,Y 370.918,Z 508.871,A -85,B 0,C 180,E1 17661.51,E2 17661.51} C_VEL
LIN {X 0,Y 367.522,Z 606.23,A -85,B 0,C 180,E1 17658.864,E2 17658.864} C_VEL
LIN {X 0,Y 366.94,Z 622.631,A -85,B 0,C 180,E1 17658.139,E2 17658.139} C_VEL
LIN {X 0,Y 366.154,Z 639.018,A -85,B 0,C 180,E1 17657.108,E2 17657.108} C_VEL
LIN {X 0,Y 365.219,Z 654.479,A -85,B 0,C 180,E1 17655.807,E2 17655.807} C_VEL
LIN {X 0,Y 364.302,Z 669.023,A -85,B 0,C 180,E1 17654.22,E2 17654.22} C_VEL
LIN {X 0,Y 363.494,Z 681.097,A -85,B 0,C 180,E1 17652.551,E2 17652.551} C_VEL
LIN {X 0,Y 362.833,Z 691.367,A -85,B 0,C 180,E1 17650.801,E2 17650.801} C_VEL
LIN {X 0,Y 362.266,Z 700.995,A -85,B 0,C 180,E1 17648.732,E2 17648.732} C_VEL
LIN {X 0,Y 361.911,Z 708.442,A -85,B 0,C 180,E1 17646.663,E2 17646.663} C_VEL
LIN {X 0,Y 361.724,Z 714.487,A -85,B 0,C 180,E1 17644.439,E2 17644.439} C_VEL
LIN {X 0,Y 361.724,Z 718.822,A -85,B 0,C 180,E1 17642.06,E2 17642.06} C_VEL
LIN {X 0,Y 361.883,Z 721.117,A -85,B 0,C 180,E1 17639.842,E2 17639.842} C_VEL
LIN {X 0,Y 362.239,Z 721.709,A -85,B 0,C 180,E1 17637.469,E2 17637.469} C_VEL
LIN {X 0,Y 362.748,Z 720.502,A -85,B 0,C 180,E1 17635.257,E2 17635.257} C_VEL
LIN {X 0,Y 363.557,Z 717.335,A -85,B 0,C 180,E1 17632.891,E2 17632.891} C_VEL
LIN {X 0,Y 364.547,Z 712.456,A -85,B 0,C 180,E1 17630.688,E2 17630.688} C_VEL
LIN {X 0,Y 365.834,Z 705.603,A -85,B 0,C 180,E1 17628.492,E2 17628.492} C_VEL
LIN {X 0,Y 367.307,Z 697.128,A -85,B 0,C 180,E1 17626.461,E2 17626.461} C_VEL
LIN {X 0,Y 368.913,Z 687.131,A -85,B 0,C 180,E1 17624.597,E2 17624.597} C_VEL
LIN {X 0,Y 370.704,Z 675.222,A -85,B 0,C 180,E1 17622.822,E2 17622.822} C_VEL
LIN {X 0,Y 372.547,Z 661.408,A -85,B 0,C 180,E1 17621.213,E2 17621.213} C_VEL
LIN {X 0,Y 374.475,Z 645.604,A -85,B 0,C 180,E1 17619.771,E2 17619.771} C_VEL
LIN {X 0,Y 376.135,Z 629.362,A -85,B 0,C 180,E1 17618.643,E2 17618.643} C_VEL
LIN {X 0,Y 377.636,Z 611.667,A -85,B 0,C 180,E1 17617.742,E2 17617.742} C_VEL
LIN {X 0,Y 386.571,Z 527.18,A -85,B 0,C 180,E1 17614.522,E2 17614.522} C_VEL
LIN {X 0,Y 387.743,Z 516.01,A -85,B 0,C 180,E1 17614.079,E2 17614.079} C_VEL
LIN {X 0,Y 385.922,Z 498.117,A -85,B 0,C 180,E1 17612.678,E2 17612.678} C_VEL
LIN {X 0,Y 383.455,Z 480.847,A -85,B 0,C 180,E1 17611.031,E2 17611.031} C_VEL
LIN {X 0,Y 383.091,Z 477.2,A -85,B 0,C 180,E1 17610.615,E2 17610.615} C_VEL
LIN {X 0,Y 389.459,Z 457.364,A -85,B 0,C 180,E1 17606.674,E2 17606.674} C_VEL
LIN {X 0,Y 391.394,Z 452.318,A -85,B 0,C 180,E1 17605.603,E2 17605.603} C_VEL
LIN {X 0,Y 391.298,Z 446.675,A -85,B 0,C 180,E1 17603.279,E2 17603.279} C_VEL
LIN {X 0,Y 391.217,Z 442.789,A -85,B 0,C 180,E1 17600.856,E2 17600.856} C_VEL
LIN {X 0,Y 391.273,Z 441.418,A -85,B 0,C 180,E1 17599.336,E2 17599.336} C_VEL
LIN {X 0,Y 391.995,Z 440.496,A -85,B 0,C 180,E1 17596.876,E2 17596.876} C_VEL
LIN {X 0,Y 392.339,Z 442.244,A -85,B 0,C 180,E1 17594.682,E2 17594.682} C_VEL
LIN {X 0,Y 393.035,Z 444.401,A -85,B 0,C 180,E1 17593.104,E2 17593.104} C_VEL
LIN {X 0,Y 394.016,Z 448.175,A -85,B 0,C 180,E1 17591.283,E2 17591.283} C_VEL
LIN {X 0,Y 394.711,Z 452.656,A -85,B 0,C 180,E1 17589.764,E2 17589.764} C_VEL
LIN {X 0,Y 388.406,Z 470.845,A -85,B 0,C 180,E1 17587.164,E2 17587.164} C_VEL
LIN {X 0,Y 389.549,Z 484.498,A -85,B 0,C 180,E1 17586.284,E2 17586.284} C_VEL
LIN {X 0,Y 389.64,Z 497.316,A -85,B 0,C 180,E1 17585.684,E2 17585.684} C_VEL
LIN {X 0,Y 383.262,Z 581.572,A -85,B 0,C 180,E1 17583.287,E2 17583.287} C_VEL
LIN {X 0,Y 378.895,Z 658.485,A -85,B 0,C 180,E1 17581.242,E2 17581.242} C_VEL
LIN {X 0,Y 377.026,Z 678.31,A -85,B 0,C 180,E1 17580.444,E2 17580.444} C_VEL
LIN {X 0,Y 374.889,Z 695.935,A -85,B 0,C 180,E1 17579.461,E2 17579.461} C_VEL
LIN {X 0,Y 372.396,Z 714.234,A -85,B 0,C 180,E1 17578.113,E2 17578.113} C_VEL
LIN {X 0,Y 368.853,Z 741.857,A -85,B 0,C 180,E1 17575.618,E2 17575.618} C_VEL
LIN {X 0,Y 366.828,Z 758.168,A -85,B 0,C 180,E1 17573.791,E2 17573.791} C_VEL
LIN {X 0,Y 364.974,Z 773.01,A -85,B 0,C 180,E1 17571.767,E2 17571.767} C_VEL
LIN {X 0,Y 363.306,Z 786.964,A -85,B 0,C 180,E1 17569.451,E2 17569.451} C_VEL
LIN {X 0,Y 361.986,Z 798.968,A -85,B 0,C 180,E1 17567.025,E2 17567.025} C_VEL
LIN {X 0,Y 361.052,Z 809.422,A -85,B 0,C 180,E1 17564.432,E2 17564.432} C_VEL
LIN {X 0,Y 360.463,Z 818.15,A -85,B 0,C 180,E1 17561.719,E2 17561.719} C_VEL
LIN {X 0,Y 360.222,Z 825.014,A -85,B 0,C 180,E1 17558.942,E2 17558.942} C_VEL
LIN {X 0,Y 360.212,Z 829.929,A -85,B 0,C 180,E1 17556.215,E2 17556.215} C_VEL
LIN {X 0,Y 360.268,Z 833.102,A -85,B 0,C 180,E1 17553.501,E2 17553.501} C_VEL
LIN {X 0,Y 360.332,Z 834.594,A -85,B 0,C 180,E1 17550.795,E2 17550.795} C_VEL
LIN {X 0,Y 360.296,Z 834.432,A -85,B 0,C 180,E1 17548.092,E2 17548.092} C_VEL
LIN {X 0,Y 360.213,Z 832.643,A -85,B 0,C 180,E1 17545.383,E2 17545.383} C_VEL
LIN {X 0,Y 360.173,Z 829.219,A -85,B 0,C 180,E1 17542.663,E2 17542.663} C_VEL
LIN {X 0,Y 360.275,Z 824.11,A -85,B 0,C 180,E1 17539.93,E2 17539.93} C_VEL
LIN {X 0,Y 360.698,Z 817.213,A -85,B 0,C 180,E1 17537.187,E2 17537.187} C_VEL
LIN {X 0,Y 361.53,Z 808.372,A -85,B 0,C 180,E1 17534.439,E2 17534.439} C_VEL
LIN {X 0,Y 362.799,Z 798.045,A -85,B 0,C 180,E1 17531.855,E2 17531.855} C_VEL
LIN {X 0,Y 364.612,Z 785.503,A -85,B 0,C 180,E1 17529.283,E2 17529.283} C_VEL
LIN {X 0,Y 366.848,Z 771.23,A -85,B 0,C 180,E1 17526.891,E2 17526.891} C_VEL
LIN {X 0,Y 369.375,Z 755.833,A -85,B 0,C 180,E1 17524.765,E2 17524.765} C_VEL
LIN {X 0,Y 372.195,Z 738.807,A -85,B 0,C 180,E1 17522.826,E2 17522.826} C_VEL
LIN {X 0,Y 375.196,Z 720.332,A -85,B 0,C 180,E1 17521.117,E2 17521.117} C_VEL
LIN {X 0,Y 378.065,Z 701.827,A -85,B 0,C 180,E1 17519.745,E2 17519.745} C_VEL
LIN {X 0,Y 380.901,Z 681.816,A -85,B 0,C 180,E1 17518.596,E2 17518.596} C_VEL
LIN {X 0,Y 383.619,Z 659.718,A -85,B 0,C 180,E1 17517.659,E2 17517.659} C_VEL
LIN {X 0,Y 392.185,Z 571.144,A -85,B 0,C 180,E1 17514.857,E2 17514.857} C_VEL
LIN {X 0,Y 401.378,Z 497.43,A -85,B 0,C 180,E1 17512.422,E2 17512.422} C_VEL
LIN {X 0,Y 402.836,Z 470.564,A -85,B 0,C 180,E1 17510.785,E2 17510.785} C_VEL
LIN {X 0,Y 404.228,Z 450.242,A -85,B 0,C 180,E1 17509.348,E2 17509.348} C_VEL
LIN {X 0,Y 403.343,Z 437.981,A -85,B 0,C 180,E1 17507.103,E2 17507.103} C_VEL
LIN {X 0,Y 403.34,Z 436.714,A -85,B 0,C 180,E1 17506.787,E2 17506.787} C_VEL
LIN {X 0,Y 402.436,Z 435.934,A -85,B 0,C 180,E1 17505.281,E2 17505.281} C_VEL
LIN {X 0,Y 402.297,Z 436.992,A -85,B 0,C 180,E1 17503.263,E2 17503.263} C_VEL
LIN {X 0,Y 402.588,Z 438.205,A -85,B 0,C 180,E1 17502.47,E2 17502.47} C_VEL
LIN {X 0,Y 403.602,Z 441.331,A -85,B 0,C 180,E1 17501.033,E2 17501.033} C_VEL
LIN {X 0,Y 405.387,Z 446.236,A -85,B 0,C 180,E1 17499.519,E2 17499.519} C_VEL
LIN {X 0,Y 407.464,Z 452.553,A -85,B 0,C 180,E1 17498.172,E2 17498.172} C_VEL
LIN {X 0,Y 396.315,Z 531.071,A -85,B 0,C 180,E1 17495.58,E2 17495.58} C_VEL
LIN {X 0,Y 388.572,Z 599.995,A -85,B 0,C 180,E1 17493.368,E2 17493.368} C_VEL
LIN {X 0,Y 385.475,Z 634.018,A -85,B 0,C 180,E1 17492.243,E2 17492.243} C_VEL
LIN {X 0,Y 383.332,Z 653.596,A -85,B 0,C 180,E1 17491.313,E2 17491.313} C_VEL
LIN {X 0,Y 380.828,Z 672.93,A -85,B 0,C 180,E1 17490.097,E2 17490.097} C_VEL
LIN {X 0,Y 378.171,Z 690.818,A -85,B 0,C 180,E1 17488.669,E2 17488.669} C_VEL
LIN {X 0,Y 375.396,Z 707.533,A -85,B 0,C 180,E1 17487.008,E2 17487.008} C_VEL
LIN {X 0,Y 372.58,Z 723.328,A -85,B 0,C 180,E1 17485.088,E2 17485.088} C_VEL
LIN {X 0,Y 369.831,Z 738.002,A -85,B 0,C 180,E1 17482.912,E2 17482.912} C_VEL
LIN {X 0,Y 367.342,Z 751.017,A -85,B 0,C 180,E1 17480.556,E2 17480.556} C_VEL
LIN {X 0,Y 365.171,Z 762.37,A -85,B 0,C 180,E1 17478.023,E2 17478.023} C_VEL
LIN {X 0,Y 363.473,Z 771.601,A -85,B 0,C 180,E1 17475.476,E2 17475.476} C_VEL
LIN {X 0,Y 362.14,Z 779.405,A -85,B 0,C 180,E1 17472.76,E2 17472.76} C_VEL
LIN {X 0,Y 361.189,Z 785.68,A -85,B 0,C 180,E1 17469.882,E2 17469.882} C_VEL
LIN {X 0,Y 360.611,Z 790.144,A -85,B 0,C 180,E1 17466.963,E2 17466.963} C_VEL
LIN {X 0,Y 360.318,Z 792.745,A -85,B 0,C 180,E1 17464.137,E2 17464.137} C_VEL
LIN {X 0,Y 360.19,Z 793.705,A -85,B 0,C 180,E1 17461.272,E2 17461.272} C_VEL
LIN {X 0,Y 360.149,Z 792.967,A -85,B 0,C 180,E1 17458.409,E2 17458.409} C_VEL
LIN {X 0,Y 360.194,Z 790.524,A -85,B 0,C 180,E1 17455.542,E2 17455.542} C_VEL
LIN {X 0,Y 360.368,Z 786.588,A -85,B 0,C 180,E1 17452.827,E2 17452.827} C_VEL
LIN {X 0,Y 360.734,Z 780.978,A -85,B 0,C 180,E1 17450.105,E2 17450.105} C_VEL
LIN {X 0,Y 361.378,Z 773.548,A -85,B 0,C 180,E1 17447.374,E2 17447.374} C_VEL
LIN {X 0,Y 362.307,Z 764.679,A -85,B 0,C 180,E1 17444.801,E2 17444.801} C_VEL
LIN {X 0,Y 363.613,Z 753.722,A -85,B 0,C 180,E1 17442.228,E2 17442.228} C_VEL
LIN {X 0,Y 365.221,Z 741.13,A -85,B 0,C 180,E1 17439.821,E2 17439.821} C_VEL
LIN {X 0,Y 367.007,Z 727.417,A -85,B 0,C 180,E1 17437.663,E2 17437.663} C_VEL
LIN {X 0,Y 368.968,Z 712.122,A -85,B 0,C 180,E1 17435.675,E2 17435.675} C_VEL
LIN {X 0,Y 370.942,Z 695.835,A -85,B 0,C 180,E1 17433.937,E2 17433.937} C_VEL
LIN {X 0,Y 372.847,Z 678.658,A -85,B 0,C 180,E1 17432.445,E2 17432.445} C_VEL
LIN {X 0,Y 374.63,Z 660.25,A -85,B 0,C 180,E1 17431.173,E2 17431.173} C_VEL
LIN {X 0,Y 376.165,Z 640.917,A -85,B 0,C 180,E1 17430.156,E2 17430.156} C_VEL
LIN {X 0,Y 377.337,Z 621.125,A -85,B 0,C 180,E1 17429.419,E2 17429.419} C_VEL
LIN {X 0,Y 385.095,Z 440.812,A -85,B 0,C 180,E1 17425.067,E2 17425.067} C_VEL
LIN {X 0,Y 384.034,Z 435.879,A -85,B 0,C 180,E1 17424.838,E2 17424.838} C_VEL
LIN {X 0,Y 372.573,Z 411.734,A -85,B 0,C 180,E1 17423.105,E2 17423.105} C_VEL
LIN {X 0,Y 365.274,Z 391.276,A -85,B 0,C 180,E1 17419.964,E2 17419.964} C_VEL
LIN {X 0,Y 361.788,Z 381.733,A -85,B 0,C 180,E1 17418.449,E2 17418.449} C_VEL
LIN {X 0,Y 361.779,Z 381.734,A -85,B 0,C 180,E1 17414.29,E2 17414.29} C_VEL
LIN {X 0,Y 361.786,Z 381.733,A -85,B 0,C 180,E1 17410.29,E2 17410.29} C_VEL
LIN {X 0,Y 361.776,Z 381.735,A -85,B 0,C 180,E1 17406.194,E2 17406.194} C_VEL
LIN {X 0,Y 361.773,Z 381.735,A -85,B 0,C 180,E1 17402.049,E2 17402.049} C_VEL
LIN {X 0,Y 361.775,Z 381.736,A -85,B 0,C 180,E1 17398.024,E2 17398.024} C_VEL
LIN {X 0,Y 361.773,Z 381.732,A -85,B 0,C 180,E1 17393.971,E2 17393.971} C_VEL
LIN {X 0,Y 361.769,Z 381.736,A -85,B 0,C 180,E1 17389.874,E2 17389.874} C_VEL
LIN {X 0,Y 361.759,Z 381.738,A -85,B 0,C 180,E1 17385.716,E2 17385.716} C_VEL
LIN {X 0,Y 361.768,Z 381.737,A -85,B 0,C 180,E1 17381.802,E2 17381.802} C_VEL
LIN {X 0,Y 361.759,Z 381.735,A -85,B 0,C 180,E1 17377.624,E2 17377.624} C_VEL
LIN {X 0,Y 361.761,Z 381.729,A -85,B 0,C 180,E1 17373.645,E2 17373.645} C_VEL
LIN {X 0,Y 361.756,Z 381.731,A -85,B 0,C 180,E1 17369.525,E2 17369.525} C_VEL
LIN {X 0,Y 361.751,Z 381.735,A -85,B 0,C 180,E1 17365.403,E2 17365.403} C_VEL
LIN {X 0,Y 361.755,Z 381.734,A -85,B 0,C 180,E1 17361.416,E2 17361.416} C_VEL
LIN {X 0,Y 361.744,Z 381.735,A -85,B 0,C 180,E1 17358.543,E2 17358.543} C_VEL
LIN {X 0,Y 360.788,Z 381.857,A -85,B 0,C 180,E1 17357.323,E2 17357.323} C_VEL
LIN {X 0,Y 356.198,Z 382.43,A -85,B 0,C 180,E1 17355.018,E2 17355.018} C_VEL
LIN {X 0,Y 353.956,Z 382.706,A -85,B 0,C 180,E1 17353.428,E2 17353.428} C_VEL
LIN {X 0,Y 353.804,Z 382.723,A -85,B 0,C 180,E1 17352.975,E2 17352.975} C_VEL
LIN {X 0,Y 353.8,Z 382.724,A -85,B 0,C 180,E1 17348.793,E2 17348.793} C_VEL
LIN {X 0,Y 353.802,Z 382.724,A -85,B 0,C 180,E1 17344.56,E2 17344.56} C_VEL
LIN {X 0,Y 353.806,Z 382.723,A -85,B 0,C 180,E1 17340.36,E2 17340.36} C_VEL
LIN {X 0,Y 353.81,Z 382.729,A -85,B 0,C 180,E1 17336.171,E2 17336.171} C_VEL
LIN {X 0,Y 353.817,Z 382.729,A -85,B 0,C 180,E1 17331.971,E2 17331.971} C_VEL
LIN {X 0,Y 353.817,Z 382.724,A -85,B 0,C 180,E1 17327.952,E2 17327.952} C_VEL
LIN {X 0,Y 353.823,Z 382.725,A -85,B 0,C 180,E1 17323.816,E2 17323.816} C_VEL
LIN {X 0,Y 353.808,Z 382.775,A -85,B 0,C 180,E1 17320.219,E2 17320.219} C_VEL
LIN {X 0,Y 359.104,Z 401.126,A -85,B 0,C 180,E1 17316.287,E2 17316.287} C_VEL
LIN {X 0,Y 363.738,Z 418.818,A -85,B 0,C 180,E1 17312.738,E2 17312.738} C_VEL
LIN {X 0,Y 365.033,Z 424.872,A -85,B 0,C 180,E1 17311.585,E2 17311.585} C_VEL
LIN {X 0,Y 361.945,Z 452.508,A -85,B 0,C 180,E1 17307.117,E2 17307.117} C_VEL
LIN {X 0,Y 359.523,Z 478.177,A -85,B 0,C 180,E1 17303.057,E2 17303.057} C_VEL
LIN {X 0,Y 363.31,Z 509.667,A -85,B 0,C 180,E1 17301.89,E2 17301.89} C_VEL
LIN {X 0,Y 359.752,Z 607.177,A -85,B 0,C 180,E1 17299.15,E2 17299.15} C_VEL
LIN {X 0,Y 359.159,Z 623.242,A -85,B 0,C 180,E1 17298.42,E2 17298.42} C_VEL
LIN {X 0,Y 358.348,Z 639.605,A -85,B 0,C 180,E1 17297.371,E2 17297.371} C_VEL
LIN {X 0,Y 357.352,Z 655.592,A -85,B 0,C 180,E1 17295.998,E2 17295.998} C_VEL
LIN {X 0,Y 356.405,Z 670.241,A -85,B 0,C 180,E1 17294.363,E2 17294.363} C_VEL
LIN {X 0,Y 355.516,Z 683.282,A -85,B 0,C 180,E1 17292.507,E2 17292.507} C_VEL
LIN {X 0,Y 354.796,Z 694.143,A -85,B 0,C 180,E1 17290.555,E2 17290.555} C_VEL
LIN {X 0,Y 354.291,Z 702.81,A -85,B 0,C 180,E1 17288.602,E2 17288.602} C_VEL
LIN {X 0,Y 353.925,Z 710.629,A -85,B 0,C 180,E1 17286.326,E2 17286.326} C_VEL
LIN {X 0,Y 353.772,Z 716.373,A -85,B 0,C 180,E1 17284.052,E2 17284.052} C_VEL
LIN {X 0,Y 353.811,Z 720.337,A -85,B 0,C 180,E1 17281.782,E2 17281.782} C_VEL
LIN {X 0,Y 354.04,Z 722.609,A -85,B 0,C 180,E1 17279.353,E2 17279.353} C_VEL
LIN {X 0,Y 354.43,Z 723.048,A -85,B 0,C 180,E1 17277.09,E2 17277.09} C_VEL
LIN {X 0,Y 355.078,Z 721.589,A -85,B 0,C 180,E1 17274.668,E2 17274.668} C_VEL
LIN {X 0,Y 355.939,Z 718.491,A -85,B 0,C 180,E1 17272.413,E2 17272.413} C_VEL
LIN {X 0,Y 357.151,Z 713.12,A -85,B 0,C 180,E1 17270.005,E2 17270.005} C_VEL
LIN {X 0,Y 358.497,Z 706.6,A -85,B 0,C 180,E1 17267.926,E2 17267.926} C_VEL
LIN {X 0,Y 360.269,Z 697.327,A -85,B 0,C 180,E1 17265.7,E2 17265.7} C_VEL
LIN {X 0,Y 362.061,Z 687.105,A -85,B 0,C 180,E1 17263.804,E2 17263.804} C_VEL
LIN {X 0,Y 364.018,Z 674.838,A -85,B 0,C 180,E1 17262.001,E2 17262.001} C_VEL
LIN {X 0,Y 365.988,Z 661.6,A -85,B 0,C 180,E1 17260.448,E2 17260.448} C_VEL
LIN {X 0,Y 368.074,Z 645.598,A -85,B 0,C 180,E1 17258.988,E2 17258.988} C_VEL
LIN {X 0,Y 369.903,Z 629.399,A -85,B 0,C 180,E1 17257.848,E2 17257.848} C_VEL
LIN {X 0,Y 371.56,Z 611.347,A -85,B 0,C 180,E1 17256.924,E2 17256.924} C_VEL
LIN {X 0,Y 382.23,Z 519.889,A -85,B 0,C 180,E1 17253.34,E2 17253.34} C_VEL
LIN {X 0,Y 382.135,Z 515.334,A -85,B 0,C 180,E1 17253.044,E2 17253.044} C_VEL
LIN {X 0,Y 380.526,Z 498.082,A -85,B 0,C 180,E1 17251.581,E2 17251.581} C_VEL
LIN {X 0,Y 378.448,Z 481.601,A -85,B 0,C 180,E1 17249.891,E2 17249.891} C_VEL
LIN {X 0,Y 377.921,Z 477.232,A -85,B 0,C 180,E1 17249.383,E2 17249.383} C_VEL
LIN {X 0,Y 385.084,Z 457.808,A -85,B 0,C 180,E1 17245.346,E2 17245.346} C_VEL
LIN {X 0,Y 385.5,Z 456.54,A -85,B 0,C 180,E1 17245.026,E2 17245.026} C_VEL
LIN {X 0,Y 385.588,Z 451.539,A -85,B 0,C 180,E1 17242.757,E2 17242.757} C_VEL
LIN {X 0,Y 385.719,Z 448.344,A -85,B 0,C 180,E1 17240.574,E2 17240.574} C_VEL
LIN {X 0,Y 385.852,Z 447.008,A -85,B 0,C 180,E1 17238.838,E2 17238.838} C_VEL
LIN {X 0,Y 386.638,Z 446.423,A -85,B 0,C 180,E1 17236.741,E2 17236.741} C_VEL
LIN {X 0,Y 387.203,Z 448.827,A -85,B 0,C 180,E1 17234.121,E2 17234.121} C_VEL
LIN {X 0,Y 388.068,Z 452.41,A -85,B 0,C 180,E1 17232.059,E2 17232.059} C_VEL
LIN {X 0,Y 388.891,Z 456.88,A -85,B 0,C 180,E1 17230.336,E2 17230.336} C_VEL
LIN {X 0,Y 383.399,Z 471.549,A -85,B 0,C 180,E1 17228.184,E2 17228.184} C_VEL
LIN {X 0,Y 384.455,Z 486.015,A -85,B 0,C 180,E1 17227.176,E2 17227.176} C_VEL
LIN {X 0,Y 384.388,Z 498.611,A -85,B 0,C 180,E1 17226.561,E2 17226.561} C_VEL
LIN {X 0,Y 377.481,Z 580.067,A -85,B 0,C 180,E1 17224.151,E2 17224.151} C_VEL
LIN {X 0,Y 372.5,Z 657.79,A -85,B 0,C 180,E1 17221.991,E2 17221.991} C_VEL
LIN {X 0,Y 370.525,Z 677.114,A -85,B 0,C 180,E1 17221.194,E2 17221.194} C_VEL
LIN {X 0,Y 368.149,Z 695.155,A -85,B 0,C 180,E1 17220.162,E2 17220.162} C_VEL
LIN {X 0,Y 365.471,Z 713.434,A -85,B 0,C 180,E1 17218.784,E2 17218.784} C_VEL
LIN {X 0,Y 362.744,Z 730.631,A -85,B 0,C 180,E1 17217.141,E2 17217.141} C_VEL
LIN {X 0,Y 359.457,Z 754.904,A -85,B 0,C 180,E1 17214.485,E2 17214.485} C_VEL
LIN {X 0,Y 357.486,Z 770.131,A -85,B 0,C 180,E1 17212.444,E2 17212.444} C_VEL
LIN {X 0,Y 355.718,Z 784.148,A -85,B 0,C 180,E1 17210.147,E2 17210.147} C_VEL
LIN {X 0,Y 354.303,Z 796.228,A -85,B 0,C 180,E1 17207.745,E2 17207.745} C_VEL
LIN {X 0,Y 353.241,Z 807.114,A -85,B 0,C 180,E1 17205.094,E2 17205.094} C_VEL
LIN {X 0,Y 352.589,Z 815.859,A -85,B 0,C 180,E1 17202.446,E2 17202.446} C_VEL
LIN {X 0,Y 352.265,Z 823.103,A -85,B 0,C 180,E1 17199.64,E2 17199.64} C_VEL
LIN {X 0,Y 352.223,Z 828.443,A -85,B 0,C 180,E1 17196.847,E2 17196.847} C_VEL
LIN {X 0,Y 352.273,Z 832.002,A -85,B 0,C 180,E1 17194.069,E2 17194.069} C_VEL
LIN {X 0,Y 352.344,Z 833.865,A -85,B 0,C 180,E1 17191.301,E2 17191.301} C_VEL
LIN {X 0,Y 352.324,Z 834.074,A -85,B 0,C 180,E1 17188.536,E2 17188.536} C_VEL
LIN {X 0,Y 352.23,Z 832.641,A -85,B 0,C 180,E1 17185.767,E2 17185.767} C_VEL
LIN {X 0,Y 352.175,Z 829.581,A -85,B 0,C 180,E1 17182.988,E2 17182.988} C_VEL
LIN {X 0,Y 352.255,Z 824.842,A -85,B 0,C 180,E1 17180.194,E2 17180.194} C_VEL
LIN {X 0,Y 352.658,Z 818.338,A -85,B 0,C 180,E1 17177.39,E2 17177.39} C_VEL
LIN {X 0,Y 353.489,Z 809.924,A -85,B 0,C 180,E1 17174.58,E2 17174.58} C_VEL
LIN {X 0,Y 354.772,Z 800.092,A -85,B 0,C 180,E1 17171.94,E2 17171.94} C_VEL
LIN {X 0,Y 356.616,Z 788.106,A -85,B 0,C 180,E1 17169.312,E2 17169.312} C_VEL
LIN {X 0,Y 358.982,Z 774.126,A -85,B 0,C 180,E1 17166.8,E2 17166.8} C_VEL
LIN {X 0,Y 361.601,Z 759.466,A -85,B 0,C 180,E1 17164.622,E2 17164.622} C_VEL
LIN {X 0,Y 364.64,Z 742.769,A -85,B 0,C 180,E1 17162.57,E2 17162.57} C_VEL
LIN {X 0,Y 367.808,Z 724.957,A -85,B 0,C 180,E1 17160.793,E2 17160.793} C_VEL
LIN {X 0,Y 371.031,Z 706.051,A -85,B 0,C 180,E1 17159.277,E2 17159.277} C_VEL
LIN {X 0,Y 374.113,Z 686.706,A -85,B 0,C 180,E1 17158.05,E2 17158.05} C_VEL
LIN {X 0,Y 377.161,Z 665.614,A -85,B 0,C 180,E1 17157.041,E2 17157.041} C_VEL
LIN {X 0,Y 380.044,Z 638.502,A -85,B 0,C 180,E1 17156.105,E2 17156.105} C_VEL
LIN {X 0,Y 387.855,Z 568.055,A -85,B 0,C 180,E1 17153.796,E2 17153.796} C_VEL
LIN {X 0,Y 397.426,Z 498.909,A -85,B 0,C 180,E1 17151.437,E2 17151.437} C_VEL
LIN {X 0,Y 399.491,Z 472.789,A -85,B 0,C 180,E1 17149.791,E2 17149.791} C_VEL
LIN {X 0,Y 401.204,Z 455.04,A -85,B 0,C 180,E1 17148.504,E2 17148.504} C_VEL
LIN {X 0,Y 401.101,Z 444.2,A -85,B 0,C 180,E1 17146.45,E2 17146.45} C_VEL
LIN {X 0,Y 400.415,Z 443.72,A -85,B 0,C 180,E1 17145.167,E2 17145.167} C_VEL
LIN {X 0,Y 400.399,Z 444.989,A -85,B 0,C 180,E1 17143.078,E2 17143.078} C_VEL
LIN {X 0,Y 401.27,Z 448.638,A -85,B 0,C 180,E1 17141.36,E2 17141.36} C_VEL
LIN {X 0,Y 402.775,Z 453.523,A -85,B 0,C 180,E1 17139.847,E2 17139.847} C_VEL
LIN {X 0,Y 403.722,Z 457.233,A -85,B 0,C 180,E1 17139.062,E2 17139.062} C_VEL
LIN {X 0,Y 391.354,Z 536.658,A -85,B 0,C 180,E1 17136.395,E2 17136.395} C_VEL
LIN {X 0,Y 382.919,Z 605.078,A -85,B 0,C 180,E1 17134.124,E2 17134.124} C_VEL
LIN {X 0,Y 379.842,Z 635.318,A -85,B 0,C 180,E1 17133.073,E2 17133.073} C_VEL
LIN {X 0,Y 377.406,Z 655.27,A -85,B 0,C 180,E1 17132.085,E2 17132.085} C_VEL
LIN {X 0,Y 374.795,Z 673.551,A -85,B 0,C 180,E1 17130.9,E2 17130.9} C_VEL
LIN {X 0,Y 371.799,Z 692.031,A -85,B 0,C 180,E1 17129.388,E2 17129.388} C_VEL
LIN {X 0,Y 368.685,Z 709.188,A -85,B 0,C 180,E1 17127.629,E2 17127.629} C_VEL
LIN {X 0,Y 365.561,Z 725.261,A -85,B 0,C 180,E1 17125.604,E2 17125.604} C_VEL
LIN {X 0,Y 362.633,Z 739.653,A -85,B 0,C 180,E1 17123.393,E2 17123.393} C_VEL
LIN {X 0,Y 359.965,Z 752.413,A -85,B 0,C 180,E1 17120.997,E2 17120.997} C_VEL
LIN {X 0,Y 357.629,Z 763.561,A -85,B 0,C 180,E1 17118.416,E2 17118.416} C_VEL
LIN {X 0,Y 355.698,Z 773.147,A -85,B 0,C 180,E1 17115.655,E2 17115.655} C_VEL
LIN {X 0,Y 354.214,Z 781.111,A -85,B 0,C 180,E1 17112.719,E2 17112.719} C_VEL
LIN {X 0,Y 353.228,Z 787.076,A -85,B 0,C 180,E1 17109.778,E2 17109.778} C_VEL
LIN {X 0,Y 352.639,Z 791.195,A -85,B 0,C 180,E1 17106.839,E2 17106.839} C_VEL
LIN {X 0,Y 352.332,Z 793.567,A -85,B 0,C 180,E1 17103.905,E2 17103.905} C_VEL
LIN {X 0,Y 352.201,Z 794.244,A -85,B 0,C 180,E1 17100.976,E2 17100.976} C_VEL
LIN {X 0,Y 352.161,Z 793.212,A -85,B 0,C 180,E1 17098.031,E2 17098.031} C_VEL
LIN {X 0,Y 352.226,Z 790.479,A -85,B 0,C 180,E1 17095.115,E2 17095.115} C_VEL
LIN {X 0,Y 352.446,Z 785.927,A -85,B 0,C 180,E1 17092.173,E2 17092.173} C_VEL
LIN {X 0,Y 352.882,Z 779.869,A -85,B 0,C 180,E1 17089.387,E2 17089.387} C_VEL
LIN {X 0,Y 353.64,Z 771.808,A -85,B 0,C 180,E1 17086.559,E2 17086.559} C_VEL
LIN {X 0,Y 354.692,Z 762.499,A -85,B 0,C 180,E1 17083.963,E2 17083.963} C_VEL
LIN {X 0,Y 356.155,Z 750.867,A -85,B 0,C 180,E1 17081.334,E2 17081.334} C_VEL
LIN {X 0,Y 357.902,Z 737.814,A -85,B 0,C 180,E1 17078.922,E2 17078.922} C_VEL
LIN {X 0,Y 359.82,Z 723.62,A -85,B 0,C 180,E1 17076.76,E2 17076.76} C_VEL
LIN {X 0,Y 361.856,Z 708.161,A -85,B 0,C 180,E1 17074.816,E2 17074.816} C_VEL
LIN {X 0,Y 363.864,Z 691.718,A -85,B 0,C 180,E1 17073.126,E2 17073.126} C_VEL
LIN {X 0,Y 365.832,Z 673.95,A -85,B 0,C 180,E1 17071.651,E2 17071.651} C_VEL
LIN {X 0,Y 367.623,Z 655.103,A -85,B 0,C 180,E1 17070.419,E2 17070.419} C_VEL
LIN {X 0,Y 369.114,Z 635.491,A -85,B 0,C 180,E1 17069.455,E2 17069.455} C_VEL
LIN {X 0,Y 370.257,Z 615.403,A -85,B 0,C 180,E1 17068.769,E2 17068.769} C_VEL
LIN {X 0,Y 378.093,Z 442.124,A -85,B 0,C 180,E1 17064.506,E2 17064.506} C_VEL
LIN {X 0,Y 377.17,Z 438.609,A -85,B 0,C 180,E1 17064.323,E2 17064.323} C_VEL
LIN {X 0,Y 364.464,Z 411.883,A -85,B 0,C 180,E1 17062.323,E2 17062.323} C_VEL
LIN {X 0,Y 357.031,Z 391.578,A -85,B 0,C 180,E1 17059.125,E2 17059.125} C_VEL
LIN {X 0,Y 353.807,Z 382.727,A -85,B 0,C 180,E1 17057.663,E2 17057.663} C_VEL
LIN {X 0,Y 353.805,Z 382.726,A -85,B 0,C 180,E1 17053.424,E2 17053.424} C_VEL
LIN {X 0,Y 353.804,Z 382.725,A -85,B 0,C 180,E1 17049.255,E2 17049.255} C_VEL
LIN {X 0,Y 353.805,Z 382.727,A -85,B 0,C 180,E1 17045.206,E2 17045.206} C_VEL
LIN {X 0,Y 353.807,Z 382.726,A -85,B 0,C 180,E1 17041.098,E2 17041.098} C_VEL
LIN {X 0,Y 353.806,Z 382.724,A -85,B 0,C 180,E1 17037.064,E2 17037.064} C_VEL
LIN {X 0,Y 353.809,Z 382.723,A -85,B 0,C 180,E1 17032.887,E2 17032.887} C_VEL
LIN {X 0,Y 353.813,Z 382.725,A -85,B 0,C 180,E1 17028.791,E2 17028.791} C_VEL
LIN {X 0,Y 353.808,Z 382.726,A -85,B 0,C 180,E1 17024.735,E2 17024.735} C_VEL
LIN {X 0,Y 353.815,Z 382.725,A -85,B 0,C 180,E1 17020.585,E2 17020.585} C_VEL
LIN {X 0,Y 353.818,Z 382.723,A -85,B 0,C 180,E1 17016.49,E2 17016.49} C_VEL
LIN {X 0,Y 353.826,Z 382.719,A -85,B 0,C 180,E1 17012.267,E2 17012.267} C_VEL
LIN {X 0,Y 353.826,Z 382.716,A -85,B 0,C 180,E1 17008.219,E2 17008.219} C_VEL
LIN {X 0,Y 353.841,Z 382.723,A -85,B 0,C 180,E1 17003.999,E2 17003.999} C_VEL
LIN {X 0,Y 353.837,Z 382.724,A -85,B 0,C 180,E1 16999.91,E2 16999.91} C_VEL
LIN {X 0,Y 353.848,Z 382.724,A -85,B 0,C 180,E1 16995.745,E2 16995.745} C_VEL
LIN {X 0,Y 353.804,Z 382.723,A -85,B 0,C 180,E1 16992.975,E2 16992.975} C_VEL
LIN {X 0,Y 352.815,Z 382.853,A -85,B 0,C 180,E1 16991.728,E2 16991.728} C_VEL
LIN {X 0,Y 348.107,Z 383.441,A -85,B 0,C 180,E1 16989.281,E2 16989.281} C_VEL
LIN {X 0,Y 345.991,Z 383.703,A -85,B 0,C 180,E1 16987.651,E2 16987.651} C_VEL
LIN {X 0,Y 345.88,Z 383.713,A -85,B 0,C 180,E1 16987.28,E2 16987.28} C_VEL
LIN {X 0,Y 345.876,Z 383.712,A -85,B 0,C 180,E1 16983.194,E2 16983.194} C_VEL
LIN {X 0,Y 345.872,Z 383.716,A -85,B 0,C 180,E1 16979.031,E2 16979.031} C_VEL
LIN {X 0,Y 345.867,Z 383.719,A -85,B 0,C 180,E1 16974.88,E2 16974.88} C_VEL
LIN {X 0,Y 345.863,Z 383.718,A -85,B 0,C 180,E1 16970.72,E2 16970.72} C_VEL
LIN {X 0,Y 345.861,Z 383.716,A -85,B 0,C 180,E1 16966.521,E2 16966.521} C_VEL
LIN {X 0,Y 345.863,Z 383.718,A -85,B 0,C 180,E1 16962.262,E2 16962.262} C_VEL
LIN {X 0,Y 345.897,Z 383.905,A -85,B 0,C 180,E1 16960.864,E2 16960.864} C_VEL
LIN {X 0,Y 351.167,Z 402.138,A -85,B 0,C 180,E1 16956.862,E2 16956.862} C_VEL
LIN {X 0,Y 355.944,Z 420.127,A -85,B 0,C 180,E1 16953.165,E2 16953.165} C_VEL
LIN {X 0,Y 357.409,Z 427.024,A -85,B 0,C 180,E1 16951.826,E2 16951.826} C_VEL
LIN {X 0,Y 354.257,Z 453.964,A -85,B 0,C 180,E1 16947.391,E2 16947.391} C_VEL
LIN {X 0,Y 351.868,Z 477.986,A -85,B 0,C 180,E1 16943.517,E2 16943.517} C_VEL
LIN {X 0,Y 355.707,Z 510.548,A -85,B 0,C 180,E1 16942.28,E2 16942.28} C_VEL
LIN {X 0,Y 352.002,Z 607.821,A -85,B 0,C 180,E1 16939.46,E2 16939.46} C_VEL
LIN {X 0,Y 351.354,Z 624.569,A -85,B 0,C 180,E1 16938.672,E2 16938.672} C_VEL
LIN {X 0,Y 350.514,Z 640.762,A -85,B 0,C 180,E1 16937.6,E2 16937.6} C_VEL
LIN {X 0,Y 349.486,Z 656.64,A -85,B 0,C 180,E1 16936.197,E2 16936.197} C_VEL
LIN {X 0,Y 348.517,Z 671.154,A -85,B 0,C 180,E1 16934.539,E2 16934.539} C_VEL
LIN {X 0,Y 347.564,Z 684.759,A -85,B 0,C 180,E1 16932.554,E2 16932.554} C_VEL
LIN {X 0,Y 346.804,Z 695.997,A -85,B 0,C 180,E1 16930.465,E2 16930.465} C_VEL
LIN {X 0,Y 346.308,Z 704.522,A -85,B 0,C 180,E1 16928.468,E2 16928.468} C_VEL
LIN {X 0,Y 345.958,Z 712.291,A -85,B 0,C 180,E1 16926.139,E2 16926.139} C_VEL
LIN {X 0,Y 345.837,Z 718.299,A -85,B 0,C 180,E1 16923.647,E2 16923.647} C_VEL
LIN {X 0,Y 345.909,Z 722.005,A -85,B 0,C 180,E1 16921.325,E2 16921.325} C_VEL
LIN {X 0,Y 346.208,Z 724.124,A -85,B 0,C 180,E1 16918.842,E2 16918.842} C_VEL
LIN {X 0,Y 346.675,Z 724.315,A -85,B 0,C 180,E1 16916.528,E2 16916.528} C_VEL
LIN {X 0,Y 347.449,Z 722.702,A -85,B 0,C 180,E1 16914.054,E2 16914.054} C_VEL
LIN {X 0,Y 348.437,Z 719.384,A -85,B 0,C 180,E1 16911.751,E2 16911.751} C_VEL
LIN {X 0,Y 349.727,Z 714.253,A -85,B 0,C 180,E1 16909.457,E2 16909.457} C_VEL
LIN {X 0,Y 351.348,Z 707.089,A -85,B 0,C 180,E1 16907.175,E2 16907.175} C_VEL
LIN {X 0,Y 353.174,Z 698.359,A -85,B 0,C 180,E1 16905.071,E2 16905.071} C_VEL
LIN {X 0,Y 355.327,Z 687.204,A -85,B 0,C 180,E1 16902.984,E2 16902.984} C_VEL
LIN {X 0,Y 357.488,Z 674.695,A -85,B 0,C 180,E1 16901.153,E2 16901.153} C_VEL
LIN {X 0,Y 359.77,Z 660.443,A -85,B 0,C 180,E1 16899.502,E2 16899.502} C_VEL
LIN {X 0,Y 361.816,Z 645.965,A -85,B 0,C 180,E1 16898.181,E2 16898.181} C_VEL
LIN {X 0,Y 363.927,Z 628.678,A -85,B 0,C 180,E1 16896.96,E2 16896.96} C_VEL
LIN {X 0,Y 365.746,Z 610.703,A -85,B 0,C 180,E1 16896.038,E2 16896.038} C_VEL
LIN {X 0,Y 377.117,Z 519.923,A -85,B 0,C 180,E1 16892.356,E2 16892.356} C_VEL
LIN {X 0,Y 375.932,Z 503.22,A -85,B 0,C 180,E1 16890.918,E2 16890.918} C_VEL
LIN {X 0,Y 374.278,Z 486.797,A -85,B 0,C 180,E1 16889.198,E2 16889.198} C_VEL
LIN {X 0,Y 373.323,Z 476.84,A -85,B 0,C 180,E1 16887.975,E2 16887.975} C_VEL
LIN {X 0,Y 379.721,Z 461.336,A -85,B 0,C 180,E1 16884.599,E2 16884.599} C_VEL
LIN {X 0,Y 379.971,Z 456.742,A -85,B 0,C 180,E1 16882.375,E2 16882.375} C_VEL
LIN {X 0,Y 380.298,Z 453.701,A -85,B 0,C 180,E1 16880.095,E2 16880.095} C_VEL
LIN {X 0,Y 381.179,Z 452.323,A -85,B 0,C 180,E1 16877,E2 16877} C_VEL
LIN {X 0,Y 381.503,Z 453.876,A -85,B 0,C 180,E1 16874.958,E2 16874.958} C_VEL
LIN {X 0,Y 382.093,Z 456.015,A -85,B 0,C 180,E1 16873.326,E2 16873.326} C_VEL
LIN {X 0,Y 382.917,Z 460.138,A -85,B 0,C 180,E1 16871.348,E2 16871.348} C_VEL
LIN {X 0,Y 382.918,Z 461.631,A -85,B 0,C 180,E1 16870.851,E2 16870.851} C_VEL
LIN {X 0,Y 378.757,Z 471.984,A -85,B 0,C 180,E1 16869.293,E2 16869.293} C_VEL
LIN {X 0,Y 379.664,Z 487.623,A -85,B 0,C 180,E1 16868.112,E2 16868.112} C_VEL
LIN {X 0,Y 379.413,Z 500.003,A -85,B 0,C 180,E1 16867.482,E2 16867.482} C_VEL
LIN {X 0,Y 371.982,Z 578.148,A -85,B 0,C 180,E1 16865.08,E2 16865.08} C_VEL
LIN {X 0,Y 366.272,Z 657.167,A -85,B 0,C 180,E1 16862.785,E2 16862.785} C_VEL
LIN {X 0,Y 364.194,Z 675.811,A -85,B 0,C 180,E1 16861.996,E2 16861.996} C_VEL
LIN {X 0,Y 361.64,Z 693.815,A -85,B 0,C 180,E1 16860.948,E2 16860.948} C_VEL
LIN {X 0,Y 358.913,Z 711.065,A -85,B 0,C 180,E1 16859.638,E2 16859.638} C_VEL
LIN {X 0,Y 355.961,Z 728.354,A -85,B 0,C 180,E1 16857.975,E2 16857.975} C_VEL
LIN {X 0,Y 353.121,Z 744.673,A -85,B 0,C 180,E1 16856.033,E2 16856.033} C_VEL
LIN {X 0,Y 350.49,Z 763.65,A -85,B 0,C 180,E1 16853.629,E2 16853.629} C_VEL
LIN {X 0,Y 348.606,Z 777.815,A -85,B 0,C 180,E1 16851.45,E2 16851.45} C_VEL
LIN {X 0,Y 346.961,Z 790.915,A -85,B 0,C 180,E1 16849.004,E2 16849.004} C_VEL
LIN {X 0,Y 345.708,Z 802.083,A -85,B 0,C 180,E1 16846.466,E2 16846.466} C_VEL
LIN {X 0,Y 344.863,Z 811.769,A -85,B 0,C 180,E1 16843.753,E2 16843.753} C_VEL
LIN {X 0,Y 344.381,Z 819.453,A -85,B 0,C 180,E1 16841.048,E2 16841.048} C_VEL
LIN {X 0,Y 344.231,Z 825.684,A -85,B 0,C 180,E1 16838.183,E2 16838.183} C_VEL
LIN {X 0,Y 344.255,Z 830.069,A -85,B 0,C 180,E1 16835.333,E2 16835.333} C_VEL
LIN {X 0,Y 344.334,Z 832.711,A -85,B 0,C 180,E1 16832.496,E2 16832.496} C_VEL
LIN {X 0,Y 344.36,Z 833.674,A -85,B 0,C 180,E1 16829.667,E2 16829.667} C_VEL
LIN {X 0,Y 344.276,Z 832.982,A -85,B 0,C 180,E1 16826.837,E2 16826.837} C_VEL
LIN {X 0,Y 344.187,Z 830.655,A -85,B 0,C 180,E1 16823.997,E2 16823.997} C_VEL
LIN {X 0,Y 344.195,Z 826.677,A -85,B 0,C 180,E1 16821.143,E2 16821.143} C_VEL
LIN {X 0,Y 344.486,Z 820.99,A -85,B 0,C 180,E1 16818.277,E2 16818.277} C_VEL
LIN {X 0,Y 345.207,Z 813.479,A -85,B 0,C 180,E1 16815.405,E2 16815.405} C_VEL
LIN {X 0,Y 346.455,Z 803.978,A -85,B 0,C 180,E1 16812.534,E2 16812.534} C_VEL
LIN {X 0,Y 348.225,Z 792.986,A -85,B 0,C 180,E1 16809.845,E2 16809.845} C_VEL
LIN {X 0,Y 350.619,Z 779.701,A -85,B 0,C 180,E1 16807.18,E2 16807.18} C_VEL
LIN {X 0,Y 353.407,Z 765.247,A -85,B 0,C 180,E1 16804.799,E2 16804.799} C_VEL
LIN {X 0,Y 356.581,Z 749.253,A -85,B 0,C 180,E1 16802.622,E2 16802.622} C_VEL
LIN {X 0,Y 360.059,Z 731.454,A -85,B 0,C 180,E1 16800.651,E2 16800.651} C_VEL
LIN {X 0,Y 363.641,Z 712.597,A -85,B 0,C 180,E1 16798.965,E2 16798.965} C_VEL
LIN {X 0,Y 367.218,Z 692.821,A -85,B 0,C 180,E1 16797.561,E2 16797.561} C_VEL
LIN {X 0,Y 370.609,Z 672.143,A -85,B 0,C 180,E1 16796.445,E2 16796.445} C_VEL
LIN {X 0,Y 373.749,Z 648.563,A -85,B 0,C 180,E1 16795.512,E2 16795.512} C_VEL
LIN {X 0,Y 382.188,Z 577.967,A -85,B 0,C 180,E1 16793.124,E2 16793.124} C_VEL
LIN {X 0,Y 393.781,Z 501.543,A -85,B 0,C 180,E1 16790.478,E2 16790.478} C_VEL
LIN {X 0,Y 396.507,Z 475.645,A -85,B 0,C 180,E1 16788.804,E2 16788.804} C_VEL
LIN {X 0,Y 398.531,Z 459.83,A -85,B 0,C 180,E1 16787.628,E2 16787.628} C_VEL
LIN {X 0,Y 398.821,Z 451.648,A -85,B 0,C 180,E1 16786.015,E2 16786.015} C_VEL
LIN {X 0,Y 398.253,Z 451.716,A -85,B 0,C 180,E1 16784.519,E2 16784.519} C_VEL
LIN {X 0,Y 398.351,Z 452.887,A -85,B 0,C 180,E1 16783.155,E2 16783.155} C_VEL
LIN {X 0,Y 399.017,Z 456.164,A -85,B 0,C 180,E1 16781.608,E2 16781.608} C_VEL
LIN {X 0,Y 400.218,Z 460.906,A -85,B 0,C 180,E1 16780.167,E2 16780.167} C_VEL
LIN {X 0,Y 400.298,Z 461.919,A -85,B 0,C 180,E1 16780,E2 16780} C_VEL
LIN {X 0,Y 386.911,Z 540.698,A -85,B 0,C 180,E1 16777.3,E2 16777.3} C_VEL
LIN {X 0,Y 377.684,Z 608.608,A -85,B 0,C 180,E1 16774.976,E2 16774.976} C_VEL
LIN {X 0,Y 374.48,Z 636.62,A -85,B 0,C 180,E1 16773.954,E2 16773.954} C_VEL
LIN {X 0,Y 371.906,Z 655.644,A -85,B 0,C 180,E1 16772.985,E2 16772.985} C_VEL
LIN {X 0,Y 368.818,Z 675.325,A -85,B 0,C 180,E1 16771.673,E2 16771.673} C_VEL
LIN {X 0,Y 365.545,Z 693.541,A -85,B 0,C 180,E1 16770.127,E2 16770.127} C_VEL
LIN {X 0,Y 362.204,Z 710.411,A -85,B 0,C 180,E1 16768.346,E2 16768.346} C_VEL
LIN {X 0,Y 358.85,Z 726.265,A -85,B 0,C 180,E1 16766.297,E2 16766.297} C_VEL
LIN {X 0,Y 355.69,Z 740.486,A -85,B 0,C 180,E1 16764.054,E2 16764.054} C_VEL
LIN {X 0,Y 352.804,Z 753.145,A -85,B 0,C 180,E1 16761.618,E2 16761.618} C_VEL
LIN {X 0,Y 350.265,Z 764.228,A -85,B 0,C 180,E1 16758.991,E2 16758.991} C_VEL
LIN {X 0,Y 348.148,Z 773.768,A -85,B 0,C 180,E1 16756.175,E2 16756.175} C_VEL
LIN {X 0,Y 346.506,Z 781.698,A -85,B 0,C 180,E1 16753.177,E2 16753.177} C_VEL
LIN {X 0,Y 345.401,Z 787.641,A -85,B 0,C 180,E1 16750.171,E2 16750.171} C_VEL
LIN {X 0,Y 344.731,Z 791.742,A -85,B 0,C 180,E1 16747.164,E2 16747.164} C_VEL
LIN {X 0,Y 344.375,Z 794.1,A -85,B 0,C 180,E1 16744.162,E2 16744.162} C_VEL
LIN {X 0,Y 344.222,Z 794.762,A -85,B 0,C 180,E1 16741.165,E2 16741.165} C_VEL
LIN {X 0,Y 344.173,Z 793.722,A -85,B 0,C 180,E1 16738.169,E2 16738.169} C_VEL
LIN {X 0,Y 344.232,Z 790.959,A -85,B 0,C 180,E1 16735.168,E2 16735.168} C_VEL
LIN {X 0,Y 344.457,Z 786.378,A -85,B 0,C 180,E1 16732.159,E2 16732.159} C_VEL
LIN {X 0,Y 344.907,Z 780.285,A -85,B 0,C 180,E1 16729.308,E2 16729.308} C_VEL
LIN {X 0,Y 345.683,Z 772.294,A -85,B 0,C 180,E1 16726.45,E2 16726.45} C_VEL
LIN {X 0,Y 346.788,Z 762.817,A -85,B 0,C 180,E1 16723.759,E2 16723.759} C_VEL
LIN {X 0,Y 348.31,Z 751.121,A -85,B 0,C 180,E1 16721.072,E2 16721.072} C_VEL
LIN {X 0,Y 350.027,Z 738.702,A -85,B 0,C 180,E1 16718.729,E2 16718.729} C_VEL
LIN {X 0,Y 352.037,Z 724.303,A -85,B 0,C 180,E1 16716.481,E2 16716.481} C_VEL
LIN {X 0,Y 354.139,Z 708.883,A -85,B 0,C 180,E1 16714.497,E2 16714.497} C_VEL
LIN {X 0,Y 356.213,Z 692.514,A -85,B 0,C 180,E1 16712.772,E2 16712.772} C_VEL
LIN {X 0,Y 358.302,Z 674.26,A -85,B 0,C 180,E1 16711.225,E2 16711.225} C_VEL
LIN {X 0,Y 360.215,Z 654.765,A -85,B 0,C 180,E1 16709.932,E2 16709.932} C_VEL
LIN {X 0,Y 361.748,Z 635.185,A -85,B 0,C 180,E1 16708.959,E2 16708.959} C_VEL
LIN {X 0,Y 362.917,Z 615.044,A -85,B 0,C 180,E1 16708.267,E2 16708.267} C_VEL
LIN {X 0,Y 371.088,Z 443.285,A -85,B 0,C 180,E1 16703.924,E2 16703.924} C_VEL
LIN {X 0,Y 358.127,Z 415.92,A -85,B 0,C 180,E1 16701.871,E2 16701.871} C_VEL
LIN {X 0,Y 356.322,Z 412.124,A -85,B 0,C 180,E1 16701.526,E2 16701.526} C_VEL
LIN {X 0,Y 349.095,Z 392.452,A -85,B 0,C 180,E1 16698.357,E2 16698.357} C_VEL
LIN {X 0,Y 345.884,Z 383.714,A -85,B 0,C 180,E1 16696.878,E2 16696.878} C_VEL
LIN {X 0,Y 345.889,Z 383.712,A -85,B 0,C 180,E1 16692.757,E2 16692.757} C_VEL
LIN {X 0,Y 345.895,Z 383.714,A -85,B 0,C 180,E1 16688.637,E2 16688.637} C_VEL
LIN {X 0,Y 345.898,Z 383.713,A -85,B 0,C 180,E1 16684.31,E2 16684.31} C_VEL
LIN {X 0,Y 345.909,Z 383.712,A -85,B 0,C 180,E1 16680.196,E2 16680.196} C_VEL
LIN {X 0,Y 345.892,Z 383.713,A -85,B 0,C 180,E1 16675.973,E2 16675.973} C_VEL
LIN {X 0,Y 345.881,Z 383.711,A -85,B 0,C 180,E1 16671.717,E2 16671.717} C_VEL
LIN {X 0,Y 345.872,Z 383.709,A -85,B 0,C 180,E1 16667.497,E2 16667.497} C_VEL
LIN {X 0,Y 345.867,Z 383.709,A -85,B 0,C 180,E1 16663.372,E2 16663.372} C_VEL
LIN {X 0,Y 345.863,Z 383.709,A -85,B 0,C 180,E1 16659.149,E2 16659.149} C_VEL
LIN {X 0,Y 345.862,Z 383.711,A -85,B 0,C 180,E1 16654.975,E2 16654.975} C_VEL
LIN {X 0,Y 345.862,Z 383.713,A -85,B 0,C 180,E1 16650.828,E2 16650.828} C_VEL
LIN {X 0,Y 345.864,Z 383.708,A -85,B 0,C 180,E1 16646.685,E2 16646.685} C_VEL
LIN {X 0,Y 345.868,Z 383.708,A -85,B 0,C 180,E1 16642.525,E2 16642.525} C_VEL
LIN {X 0,Y 345.876,Z 383.712,A -85,B 0,C 180,E1 16638.325,E2 16638.325} C_VEL
LIN {X 0,Y 345.877,Z 383.715,A -85,B 0,C 180,E1 16634.232,E2 16634.232} C_VEL
LIN {X 0,Y 345.887,Z 383.715,A -85,B 0,C 180,E1 16630.056,E2 16630.056} C_VEL
LIN {X 0,Y 345.88,Z 383.713,A -85,B 0,C 180,E1 16627.28,E2 16627.28} C_VEL
LIN {X 0,Y 344.867,Z 383.838,A -85,B 0,C 180,E1 16626.004,E2 16626.004} C_VEL
LIN {X 0,Y 338.352,Z 384.658,A -85,B 0,C 180,E1 16622.209,E2 16622.209} C_VEL
LIN {X 0,Y 337.958,Z 384.702,A -85,B 0,C 180,E1 16621.452,E2 16621.452} C_VEL
LIN {X 0,Y 337.941,Z 384.708,A -85,B 0,C 180,E1 16617.218,E2 16617.218} C_VEL
LIN {X 0,Y 337.936,Z 384.708,A -85,B 0,C 180,E1 16613.022,E2 16613.022} C_VEL
LIN {X 0,Y 337.933,Z 384.703,A -85,B 0,C 180,E1 16608.94,E2 16608.94} C_VEL
LIN {X 0,Y 337.928,Z 384.705,A -85,B 0,C 180,E1 16604.756,E2 16604.756} C_VEL
LIN {X 0,Y 337.965,Z 384.746,A -85,B 0,C 180,E1 16601.592,E2 16601.592} C_VEL
LIN {X 0,Y 343.175,Z 402.864,A -85,B 0,C 180,E1 16597.513,E2 16597.513} C_VEL
LIN {X 0,Y 347.826,Z 420.375,A -85,B 0,C 180,E1 16593.823,E2 16593.823} C_VEL
LIN {X 0,Y 349.809,Z 428.875,A -85,B 0,C 180,E1 16592.117,E2 16592.117} C_VEL
LIN {X 0,Y 346.565,Z 455.505,A -85,B 0,C 180,E1 16587.66,E2 16587.66} C_VEL
LIN {X 0,Y 344.242,Z 477.919,A -85,B 0,C 180,E1 16583.988,E2 16583.988} C_VEL
LIN {X 0,Y 348.109,Z 511.421,A -85,B 0,C 180,E1 16582.681,E2 16582.681} C_VEL
LIN {X 0,Y 344.253,Z 607.917,A -85,B 0,C 180,E1 16579.787,E2 16579.787} C_VEL
LIN {X 0,Y 343.573,Z 624.838,A -85,B 0,C 180,E1 16578.975,E2 16578.975} C_VEL
LIN {X 0,Y 342.738,Z 640.527,A -85,B 0,C 180,E1 16577.925,E2 16577.925} C_VEL
LIN {X 0,Y 341.672,Z 656.668,A -85,B 0,C 180,E1 16576.491,E2 16576.491} C_VEL
LIN {X 0,Y 340.663,Z 671.391,A -85,B 0,C 180,E1 16574.794,E2 16574.794} C_VEL
LIN {X 0,Y 339.742,Z 684.207,A -85,B 0,C 180,E1 16572.925,E2 16572.925} C_VEL
LIN {X 0,Y 339.025,Z 694.565,A -85,B 0,C 180,E1 16571.052,E2 16571.052} C_VEL
LIN {X 0,Y 338.43,Z 704.358,A -85,B 0,C 180,E1 16568.838,E2 16568.838} C_VEL
LIN {X 0,Y 338.063,Z 711.929,A -85,B 0,C 180,E1 16566.624,E2 16566.624} C_VEL
LIN {X 0,Y 337.901,Z 718.102,A -85,B 0,C 180,E1 16564.243,E2 16564.243} C_VEL
LIN {X 0,Y 337.956,Z 722.611,A -85,B 0,C 180,E1 16561.696,E2 16561.696} C_VEL
LIN {X 0,Y 338.228,Z 725.043,A -85,B 0,C 180,E1 16559.323,E2 16559.323} C_VEL
LIN {X 0,Y 338.731,Z 725.798,A -85,B 0,C 180,E1 16556.785,E2 16556.785} C_VEL
LIN {X 0,Y 339.468,Z 724.768,A -85,B 0,C 180,E1 16554.422,E2 16554.422} C_VEL
LIN {X 0,Y 340.559,Z 721.76,A -85,B 0,C 180,E1 16551.899,E2 16551.899} C_VEL
LIN {X 0,Y 341.902,Z 717.131,A -85,B 0,C 180,E1 16549.554,E2 16549.554} C_VEL
LIN {X 0,Y 343.601,Z 710.547,A -85,B 0,C 180,E1 16547.223,E2 16547.223} C_VEL
LIN {X 0,Y 345.668,Z 701.73,A -85,B 0,C 180,E1 16544.911,E2 16544.911} C_VEL
LIN {X 0,Y 347.758,Z 692.089,A -85,B 0,C 180,E1 16542.947,E2 16542.947} C_VEL
LIN {X 0,Y 350.136,Z 680.072,A -85,B 0,C 180,E1 16541.002,E2 16541.002} C_VEL
LIN {X 0,Y 352.486,Z 666.9,A -85,B 0,C 180,E1 16539.32,E2 16539.32} C_VEL
LIN {X 0,Y 354.904,Z 652.174,A -85,B 0,C 180,E1 16537.82,E2 16537.82} C_VEL
LIN {X 0,Y 357.117,Z 636.511,A -85,B 0,C 180,E1 16536.574,E2 16536.574} C_VEL
LIN {X 0,Y 359.278,Z 618.663,A -85,B 0,C 180,E1 16535.502,E2 16535.502} C_VEL
LIN {X 0,Y 364.65,Z 574.757,A -85,B 0,C 180,E1 16533.612,E2 16533.612} C_VEL
LIN {X 0,Y 372.136,Z 521.902,A -85,B 0,C 180,E1 16531.429,E2 16531.429} C_VEL
LIN {X 0,Y 371.25,Z 505.2,A -85,B 0,C 180,E1 16529.915,E2 16529.915} C_VEL
LIN {X 0,Y 370.057,Z 489.763,A -85,B 0,C 180,E1 16528.206,E2 16528.206} C_VEL
LIN {X 0,Y 369.179,Z 476.515,A -85,B 0,C 180,E1 16526.462,E2 16526.462} C_VEL
LIN {X 0,Y 374.006,Z 466.062,A -85,B 0,C 180,E1 16524.1,E2 16524.1} C_VEL
LIN {X 0,Y 374.447,Z 461.893,A -85,B 0,C 180,E1 16521.916,E2 16521.916} C_VEL
LIN {X 0,Y 374.954,Z 459.234,A -85,B 0,C 180,E1 16519.61,E2 16519.61} C_VEL
LIN {X 0,Y 375.89,Z 458.288,A -85,B 0,C 180,E1 16516.789,E2 16516.789} C_VEL
LIN {X 0,Y 376.54,Z 460.955,A -85,B 0,C 180,E1 16513.978,E2 16513.978} C_VEL
LIN {X 0,Y 377.231,Z 464.936,A -85,B 0,C 180,E1 16511.858,E2 16511.858} C_VEL
LIN {X 0,Y 377.332,Z 465.902,A -85,B 0,C 180,E1 16511.488,E2 16511.488} C_VEL
LIN {X 0,Y 374.531,Z 472.548,A -85,B 0,C 180,E1 16510.462,E2 16510.462} C_VEL
LIN {X 0,Y 375.125,Z 487.982,A -85,B 0,C 180,E1 16509.19,E2 16509.19} C_VEL
LIN {X 0,Y 374.772,Z 501.051,A -85,B 0,C 180,E1 16508.459,E2 16508.459} C_VEL
LIN {X 0,Y 366.622,Z 577.822,A -85,B 0,C 180,E1 16506.013,E2 16506.013} C_VEL
LIN {X 0,Y 360.207,Z 656.895,A -85,B 0,C 180,E1 16503.618,E2 16503.618} C_VEL
LIN {X 0,Y 357.857,Z 675.989,A -85,B 0,C 180,E1 16502.775,E2 16502.775} C_VEL
LIN {X 0,Y 355.055,Z 693.954,A -85,B 0,C 180,E1 16501.682,E2 16501.682} C_VEL
LIN {X 0,Y 352.013,Z 711.548,A -85,B 0,C 180,E1 16500.29,E2 16500.29} C_VEL
LIN {X 0,Y 348.802,Z 728.929,A -85,B 0,C 180,E1 16498.552,E2 16498.552} C_VEL
LIN {X 0,Y 345.841,Z 744.488,A -85,B 0,C 180,E1 16496.623,E2 16496.623} C_VEL
LIN {X 0,Y 343.11,Z 760.409,A -85,B 0,C 180,E1 16494.352,E2 16494.352} C_VEL
LIN {X 0,Y 341.079,Z 775.099,A -85,B 0,C 180,E1 16492.129,E2 16492.129} C_VEL
LIN {X 0,Y 339.3,Z 788.637,A -85,B 0,C 180,E1 16489.63,E2 16489.63} C_VEL
LIN {X 0,Y 337.926,Z 800.137,A -85,B 0,C 180,E1 16487.033,E2 16487.033} C_VEL
LIN {X 0,Y 336.985,Z 810.121,A -85,B 0,C 180,E1 16484.257,E2 16484.257} C_VEL
LIN {X 0,Y 336.439,Z 818.07,A -85,B 0,C 180,E1 16481.485,E2 16481.485} C_VEL
LIN {X 0,Y 336.244,Z 824.54,A -85,B 0,C 180,E1 16478.551,E2 16478.551} C_VEL
LIN {X 0,Y 336.268,Z 829.145,A -85,B 0,C 180,E1 16475.631,E2 16475.631} C_VEL
LIN {X 0,Y 336.348,Z 831.991,A -85,B 0,C 180,E1 16472.726,E2 16472.726} C_VEL
LIN {X 0,Y 336.388,Z 833.136,A -85,B 0,C 180,E1 16470,E2 16470} C_VEL
LIN {X 0,Y 336.295,Z 832.726,A -85,B 0,C 180,E1 16467.103,E2 16467.103} C_VEL
LIN {X 0,Y 336.191,Z 830.673,A -85,B 0,C 180,E1 16464.196,E2 16464.196} C_VEL
LIN {X 0,Y 336.197,Z 826.693,A -85,B 0,C 180,E1 16461.103,E2 16461.103} C_VEL
LIN {X 0,Y 336.54,Z 820.803,A -85,B 0,C 180,E1 16457.997,E2 16457.997} C_VEL
LIN {X 0,Y 337.339,Z 813.404,A -85,B 0,C 180,E1 16455.057,E2 16455.057} C_VEL
LIN {X 0,Y 338.709,Z 804.036,A -85,B 0,C 180,E1 16452.121,E2 16452.121} C_VEL
LIN {X 0,Y 340.628,Z 793.227,A -85,B 0,C 180,E1 16449.375,E2 16449.375} C_VEL
LIN {X 0,Y 343.203,Z 780.15,A -85,B 0,C 180,E1 16446.658,E2 16446.658} C_VEL
LIN {X 0,Y 346.301,Z 765.473,A -85,B 0,C 180,E1 16444.152,E2 16444.152} C_VEL
LIN {X 0,Y 349.844,Z 749.15,A -85,B 0,C 180,E1 16441.863,E2 16441.863} C_VEL
LIN {X 0,Y 353.586,Z 731.731,A -85,B 0,C 180,E1 16439.872,E2 16439.872} C_VEL
LIN {X 0,Y 357.407,Z 713.383,A -85,B 0,C 180,E1 16438.174,E2 16438.174} C_VEL
LIN {X 0,Y 361.193,Z 694.274,A -85,B 0,C 180,E1 16436.763,E2 16436.763} C_VEL
LIN {X 0,Y 365.074,Z 673.142,A -85,B 0,C 180,E1 16435.559,E2 16435.559} C_VEL
LIN {X 0,Y 368.569,Z 649.845,A -85,B 0,C 180,E1 16434.589,E2 16434.589} C_VEL
LIN {X 0,Y 378.189,Z 577.765,A -85,B 0,C 180,E1 16432.065,E2 16432.065} C_VEL
LIN {X 0,Y 390.645,Z 503.252,A -85,B 0,C 180,E1 16429.425,E2 16429.425} C_VEL
LIN {X 0,Y 394.062,Z 477.805,A -85,B 0,C 180,E1 16427.736,E2 16427.736} C_VEL
LIN {X 0,Y 396.167,Z 464.761,A -85,B 0,C 180,E1 16426.747,E2 16426.747} C_VEL
LIN {X 0,Y 396.674,Z 459.193,A -85,B 0,C 180,E1 16425.61,E2 16425.61} C_VEL
LIN {X 0,Y 396.303,Z 460.108,A -85,B 0,C 180,E1 16423.606,E2 16423.606} C_VEL
LIN {X 0,Y 396.72,Z 463.405,A -85,B 0,C 180,E1 16421.97,E2 16421.97} C_VEL
LIN {X 0,Y 397.277,Z 466.631,A -85,B 0,C 180,E1 16420.967,E2 16420.967} C_VEL
LIN {X 0,Y 382.793,Z 544.929,A -85,B 0,C 180,E1 16418.24,E2 16418.24} C_VEL
LIN {X 0,Y 372.838,Z 611.372,A -85,B 0,C 180,E1 16415.9,E2 16415.9} C_VEL
LIN {X 0,Y 369.419,Z 638.006,A -85,B 0,C 180,E1 16414.885,E2 16414.885} C_VEL
LIN {X 0,Y 366.406,Z 657.956,A -85,B 0,C 180,E1 16413.826,E2 16413.826} C_VEL
LIN {X 0,Y 363.029,Z 677.278,A -85,B 0,C 180,E1 16412.484,E2 16412.484} C_VEL
LIN {X 0,Y 359.409,Z 695.434,A -85,B 0,C 180,E1 16410.882,E2 16410.882} C_VEL
LIN {X 0,Y 355.543,Z 713.215,A -85,B 0,C 180,E1 16408.927,E2 16408.927} C_VEL
LIN {X 0,Y 351.986,Z 728.594,A -85,B 0,C 180,E1 16406.85,E2 16406.85} C_VEL
LIN {X 0,Y 348.615,Z 742.414,A -85,B 0,C 180,E1 16404.574,E2 16404.574} C_VEL
LIN {X 0,Y 345.52,Z 754.731,A -85,B 0,C 180,E1 16402.098,E2 16402.098} C_VEL
LIN {X 0,Y 342.802,Z 765.598,A -85,B 0,C 180,E1 16399.421,E2 16399.421} C_VEL
LIN {X 0,Y 340.524,Z 774.955,A -85,B 0,C 180,E1 16396.548,E2 16396.548} C_VEL
LIN {X 0,Y 338.832,Z 782.342,A -85,B 0,C 180,E1 16393.655,E2 16393.655} C_VEL
LIN {X 0,Y 337.595,Z 788.247,A -85,B 0,C 180,E1 16390.581,E2 16390.581} C_VEL
LIN {X 0,Y 336.832,Z 792.329,A -85,B 0,C 180,E1 16387.494,E2 16387.494} C_VEL
LIN {X 0,Y 336.424,Z 794.65,A -85,B 0,C 180,E1 16384.432,E2 16384.432} C_VEL
LIN {X 0,Y 336.245,Z 795.287,A -85,B 0,C 180,E1 16381.363,E2 16381.363} C_VEL
LIN {X 0,Y 336.185,Z 794.22,A -85,B 0,C 180,E1 16378.295,E2 16378.295} C_VEL
LIN {X 0,Y 336.238,Z 791.426,A -85,B 0,C 180,E1 16375.224,E2 16375.224} C_VEL
LIN {X 0,Y 336.468,Z 786.806,A -85,B 0,C 180,E1 16372.143,E2 16372.143} C_VEL
LIN {X 0,Y 336.939,Z 780.572,A -85,B 0,C 180,E1 16369.186,E2 16369.186} C_VEL
LIN {X 0,Y 337.736,Z 772.622,A -85,B 0,C 180,E1 16366.3,E2 16366.3} C_VEL
LIN {X 0,Y 338.907,Z 762.915,A -85,B 0,C 180,E1 16363.503,E2 16363.503} C_VEL
LIN {X 0,Y 340.468,Z 751.31,A -85,B 0,C 180,E1 16360.797,E2 16360.797} C_VEL
LIN {X 0,Y 342.253,Z 738.809,A -85,B 0,C 180,E1 16358.401,E2 16358.401} C_VEL
LIN {X 0,Y 344.342,Z 724.317,A -85,B 0,C 180,E1 16356.105,E2 16356.105} C_VEL
LIN {X 0,Y 346.523,Z 708.777,A -85,B 0,C 180,E1 16354.078,E2 16354.078} C_VEL
LIN {X 0,Y 348.674,Z 692.256,A -85,B 0,C 180,E1 16352.318,E2 16352.318} C_VEL
LIN {X 0,Y 350.723,Z 674.953,A -85,B 0,C 180,E1 16350.824,E2 16350.824} C_VEL
LIN {X 0,Y 352.65,Z 656.039,A -85,B 0,C 180,E1 16349.534,E2 16349.534} C_VEL
LIN {X 0,Y 354.268,Z 636.285,A -85,B 0,C 180,E1 16348.517,E2 16348.517} C_VEL
LIN {X 0,Y 355.512,Z 616.115,A -85,B 0,C 180,E1 16347.794,E2 16347.794} C_VEL
LIN {X 0,Y 364.034,Z 445.482,A -85,B 0,C 180,E1 16343.353,E2 16343.353} C_VEL
LIN {X 0,Y 349.788,Z 415.772,A -85,B 0,C 180,E1 16341.033,E2 16341.033} C_VEL
LIN {X 0,Y 348.434,Z 412.882,A -85,B 0,C 180,E1 16340.786,E2 16340.786} C_VEL
LIN {X 0,Y 341.217,Z 393.557,A -85,B 0,C 180,E1 16337.598,E2 16337.598} C_VEL
LIN {X 0,Y 337.948,Z 384.702,A -85,B 0,C 180,E1 16336.081,E2 16336.081} C_VEL
LIN {X 0,Y 337.937,Z 384.702,A -85,B 0,C 180,E1 16331.789,E2 16331.789} C_VEL
LIN {X 0,Y 337.928,Z 384.705,A -85,B 0,C 180,E1 16327.537,E2 16327.537} C_VEL
LIN {X 0,Y 337.928,Z 384.705,A -85,B 0,C 180,E1 16323.139,E2 16323.139} C_VEL
LIN {X 0,Y 337.928,Z 384.701,A -85,B 0,C 180,E1 16319.028,E2 16319.028} C_VEL
LIN {X 0,Y 337.942,Z 384.702,A -85,B 0,C 180,E1 16314.726,E2 16314.726} C_VEL
LIN {X 0,Y 337.942,Z 384.699,A -85,B 0,C 180,E1 16310.615,E2 16310.615} C_VEL
LIN {X 0,Y 337.958,Z 384.698,A -85,B 0,C 180,E1 16306.324,E2 16306.324} C_VEL
LIN {X 0,Y 337.96,Z 384.698,A -85,B 0,C 180,E1 16302.126,E2 16302.126} C_VEL
LIN {X 0,Y 337.956,Z 384.698,A -85,B 0,C 180,E1 16297.822,E2 16297.822} C_VEL
LIN {X 0,Y 337.939,Z 384.695,A -85,B 0,C 180,E1 16293.562,E2 16293.562} C_VEL
LIN {X 0,Y 337.929,Z 384.697,A -85,B 0,C 180,E1 16289.322,E2 16289.322} C_VEL
LIN {X 0,Y 337.924,Z 384.702,A -85,B 0,C 180,E1 16285.078,E2 16285.078} C_VEL
LIN {X 0,Y 337.924,Z 384.701,A -85,B 0,C 180,E1 16280.806,E2 16280.806} C_VEL
LIN {X 0,Y 337.929,Z 384.701,A -85,B 0,C 180,E1 16276.482,E2 16276.482} C_VEL
LIN {X 0,Y 337.938,Z 384.701,A -85,B 0,C 180,E1 16272.257,E2 16272.257} C_VEL
LIN {X 0,Y 337.957,Z 384.701,A -85,B 0,C 180,E1 16267.93,E2 16267.93} C_VEL
LIN {X 0,Y 337.961,Z 384.7,A -85,B 0,C 180,E1 16263.655,E2 16263.655} C_VEL
LIN {X 0,Y 337.958,Z 384.702,A -85,B 0,C 180,E1 16261.452,E2 16261.452} C_VEL
LIN {X 0,Y 336.911,Z 384.83,A -85,B 0,C 180,E1 16260.147,E2 16260.147} C_VEL
LIN {X 0,Y 330.379,Z 385.648,A -85,B 0,C 180,E1 16256.261,E2 16256.261} C_VEL
LIN {X 0,Y 330.014,Z 385.695,A -85,B 0,C 180,E1 16255.486,E2 16255.486} C_VEL
LIN {X 0,Y 330.002,Z 385.696,A -85,B 0,C 180,E1 16251.14,E2 16251.14} C_VEL
LIN {X 0,Y 329.993,Z 385.692,A -85,B 0,C 180,E1 16246.905,E2 16246.905} C_VEL
LIN {X 0,Y 329.985,Z 385.696,A -85,B 0,C 180,E1 16242.508,E2 16242.508} C_VEL
LIN {X 0,Y 330.02,Z 385.94,A -85,B 0,C 180,E1 16242.268,E2 16242.268} C_VEL
LIN {X 0,Y 334.955,Z 402.681,A -85,B 0,C 180,E1 16238.382,E2 16238.382} C_VEL
LIN {X 0,Y 339.576,Z 419.98,A -85,B 0,C 180,E1 16234.63,E2 16234.63} C_VEL
LIN {X 0,Y 342.148,Z 431.235,A -85,B 0,C 180,E1 16232.329,E2 16232.329} C_VEL
LIN {X 0,Y 338.771,Z 457.845,A -85,B 0,C 180,E1 16227.796,E2 16227.796} C_VEL
LIN {X 0,Y 336.62,Z 477.882,A -85,B 0,C 180,E1 16224.465,E2 16224.465} C_VEL
LIN {X 0,Y 340.49,Z 512.303,A -85,B 0,C 180,E1 16223.081,E2 16223.081} C_VEL
LIN {X 0,Y 336.474,Z 608.825,A -85,B 0,C 180,E1 16220.087,E2 16220.087} C_VEL
LIN {X 0,Y 335.789,Z 625.251,A -85,B 0,C 180,E1 16219.28,E2 16219.28} C_VEL
LIN {X 0,Y 334.904,Z 641.348,A -85,B 0,C 180,E1 16218.179,E2 16218.179} C_VEL
LIN {X 0,Y 333.807,Z 657.515,A -85,B 0,C 180,E1 16216.712,E2 16216.712} C_VEL
LIN {X 0,Y 332.769,Z 672.293,A -85,B 0,C 180,E1 16214.975,E2 16214.975} C_VEL
LIN {X 0,Y 331.822,Z 685.164,A -85,B 0,C 180,E1 16213.062,E2 16213.062} C_VEL
LIN {X 0,Y 331.034,Z 696.246,A -85,B 0,C 180,E1 16210.996,E2 16210.996} C_VEL
LIN {X 0,Y 330.44,Z 706.03,A -85,B 0,C 180,E1 16208.702,E2 16208.702} C_VEL
LIN {X 0,Y 330.067,Z 714.047,A -85,B 0,C 180,E1 16206.261,E2 16206.261} C_VEL
LIN {X 0,Y 329.952,Z 719.974,A -85,B 0,C 180,E1 16203.823,E2 16203.823} C_VEL
LIN {X 0,Y 330.053,Z 724.114,A -85,B 0,C 180,E1 16201.389,E2 16201.389} C_VEL
LIN {X 0,Y 330.399,Z 726.567,A -85,B 0,C 180,E1 16198.786,E2 16198.786} C_VEL
LIN {X 0,Y 330.967,Z 727.194,A -85,B 0,C 180,E1 16196.363,E2 16196.363} C_VEL
LIN {X 0,Y 331.869,Z 725.939,A -85,B 0,C 180,E1 16193.774,E2 16193.774} C_VEL
LIN {X 0,Y 333.041,Z 723.088,A -85,B 0,C 180,E1 16191.367,E2 16191.367} C_VEL
LIN {X 0,Y 334.535,Z 718.389,A -85,B 0,C 180,E1 16188.972,E2 16188.972} C_VEL
LIN {X 0,Y 336.427,Z 711.837,A -85,B 0,C 180,E1 16186.596,E2 16186.596} C_VEL
LIN {X 0,Y 338.512,Z 703.7,A -85,B 0,C 180,E1 16184.408,E2 16184.408} C_VEL
LIN {X 0,Y 340.983,Z 693.436,A -85,B 0,C 180,E1 16182.245,E2 16182.245} C_VEL
LIN {X 0,Y 343.678,Z 680.921,A -85,B 0,C 180,E1 16180.188,E2 16180.188} C_VEL
LIN {X 0,Y 346.403,Z 667.193,A -85,B 0,C 180,E1 16178.407,E2 16178.407} C_VEL
LIN {X 0,Y 349.32,Z 650.634,A -85,B 0,C 180,E1 16176.734,E2 16176.734} C_VEL
LIN {X 0,Y 351.764,Z 634.504,A -85,B 0,C 180,E1 16175.481,E2 16175.481} C_VEL
LIN {X 0,Y 354.089,Z 616.283,A -85,B 0,C 180,E1 16174.426,E2 16174.426} C_VEL
LIN {X 0,Y 364.145,Z 545.641,A -85,B 0,C 180,E1 16171.382,E2 16171.382} C_VEL
LIN {X 0,Y 367.414,Z 524.049,A -85,B 0,C 180,E1 16170.469,E2 16170.469} C_VEL
LIN {X 0,Y 366.916,Z 507.922,A -85,B 0,C 180,E1 16168.932,E2 16168.932} C_VEL
LIN {X 0,Y 366.198,Z 493.245,A -85,B 0,C 180,E1 16167.233,E2 16167.233} C_VEL
LIN {X 0,Y 365.674,Z 480.779,A -85,B 0,C 180,E1 16165.528,E2 16165.528} C_VEL
LIN {X 0,Y 365.781,Z 475.945,A -85,B 0,C 180,E1 16164.777,E2 16164.777} C_VEL
LIN {X 0,Y 368.41,Z 470.8,A -85,B 0,C 180,E1 16163.533,E2 16163.533} C_VEL
LIN {X 0,Y 369.04,Z 466.972,A -85,B 0,C 180,E1 16161.288,E2 16161.288} C_VEL
LIN {X 0,Y 369.56,Z 464.961,A -85,B 0,C 180,E1 16159.249,E2 16159.249} C_VEL
LIN {X 0,Y 370.561,Z 464.268,A -85,B 0,C 180,E1 16156.737,E2 16156.737} C_VEL
LIN {X 0,Y 371.138,Z 466.973,A -85,B 0,C 180,E1 16154.003,E2 16154.003} C_VEL
LIN {X 0,Y 371.694,Z 470.544,A -85,B 0,C 180,E1 16152.079,E2 16152.079} C_VEL
LIN {X 0,Y 370.722,Z 473.028,A -85,B 0,C 180,E1 16151.708,E2 16151.708} C_VEL
LIN {X 0,Y 370.964,Z 488.05,A -85,B 0,C 180,E1 16150.357,E2 16150.357} C_VEL
LIN {X 0,Y 370.759,Z 497.28,A -85,B 0,C 180,E1 16149.742,E2 16149.742} C_VEL
LIN {X 0,Y 370.26,Z 503.654,A -85,B 0,C 180,E1 16149.432,E2 16149.432} C_VEL
LIN {X 0,Y 361.428,Z 578.743,A -85,B 0,C 180,E1 16146.961,E2 16146.961} C_VEL
LIN {X 0,Y 354.35,Z 656.575,A -85,B 0,C 180,E1 16144.503,E2 16144.503} C_VEL
LIN {X 0,Y 351.831,Z 675.176,A -85,B 0,C 180,E1 16143.653,E2 16143.653} C_VEL
LIN {X 0,Y 348.559,Z 694.434,A -85,B 0,C 180,E1 16142.44,E2 16142.44} C_VEL
LIN {X 0,Y 345.227,Z 712.055,A -85,B 0,C 180,E1 16140.987,E2 16140.987} C_VEL
LIN {X 0,Y 341.854,Z 728.914,A -85,B 0,C 180,E1 16139.239,E2 16139.239} C_VEL
LIN {X 0,Y 338.494,Z 745.019,A -85,B 0,C 180,E1 16137.153,E2 16137.153} C_VEL
LIN {X 0,Y 335.524,Z 759.576,A -85,B 0,C 180,E1 16134.846,E2 16134.846} C_VEL
LIN {X 0,Y 332.598,Z 779.235,A -85,B 0,C 180,E1 16131.613,E2 16131.613} C_VEL
LIN {X 0,Y 330.908,Z 792.011,A -85,B 0,C 180,E1 16129.046,E2 16129.046} C_VEL
LIN {X 0,Y 329.645,Z 802.869,A -85,B 0,C 180,E1 16126.385,E2 16126.385} C_VEL
LIN {X 0,Y 328.806,Z 812.264,A -85,B 0,C 180,E1 16123.541,E2 16123.541} C_VEL
LIN {X 0,Y 328.345,Z 820.063,A -85,B 0,C 180,E1 16120.528,E2 16120.528} C_VEL
LIN {X 0,Y 328.256,Z 825.878,A -85,B 0,C 180,E1 16117.526,E2 16117.526} C_VEL
LIN {X 0,Y 328.316,Z 829.865,A -85,B 0,C 180,E1 16114.542,E2 16114.542} C_VEL
LIN {X 0,Y 328.392,Z 832.114,A -85,B 0,C 180,E1 16111.57,E2 16111.57} C_VEL
LIN {X 0,Y 328.367,Z 832.664,A -85,B 0,C 180,E1 16108.604,E2 16108.604} C_VEL
LIN {X 0,Y 328.246,Z 831.536,A -85,B 0,C 180,E1 16105.633,E2 16105.633} C_VEL
LIN {X 0,Y 328.176,Z 828.774,A -85,B 0,C 180,E1 16102.648,E2 16102.648} C_VEL
LIN {X 0,Y 328.304,Z 824.36,A -85,B 0,C 180,E1 16099.642,E2 16099.642} C_VEL
LIN {X 0,Y 328.901,Z 817.854,A -85,B 0,C 180,E1 16096.463,E2 16096.463} C_VEL
LIN {X 0,Y 330.02,Z 809.811,A -85,B 0,C 180,E1 16093.454,E2 16093.454} C_VEL
LIN {X 0,Y 331.817,Z 799.78,A -85,B 0,C 180,E1 16090.459,E2 16090.459} C_VEL
LIN {X 0,Y 334.318,Z 787.659,A -85,B 0,C 180,E1 16087.539,E2 16087.539} C_VEL
LIN {X 0,Y 337.369,Z 774.05,A -85,B 0,C 180,E1 16084.863,E2 16084.863} C_VEL
LIN {X 0,Y 340.949,Z 758.793,A -85,B 0,C 180,E1 16082.397,E2 16082.397} C_VEL
LIN {X 0,Y 344.902,Z 742.139,A -85,B 0,C 180,E1 16080.187,E2 16080.187} C_VEL
LIN {X 0,Y 348.993,Z 724.702,A -85,B 0,C 180,E1 16078.292,E2 16078.292} C_VEL
LIN {X 0,Y 353.135,Z 706.312,A -85,B 0,C 180,E1 16076.682,E2 16076.682} C_VEL
LIN {X 0,Y 357.388,Z 686.233,A -85,B 0,C 180,E1 16075.296,E2 16075.296} C_VEL
LIN {X 0,Y 361.569,Z 664.398,A -85,B 0,C 180,E1 16074.157,E2 16074.157} C_VEL
LIN {X 0,Y 365.315,Z 639.626,A -85,B 0,C 180,E1 16073.191,E2 16073.191} C_VEL
LIN {X 0,Y 375.486,Z 572.651,A -85,B 0,C 180,E1 16070.777,E2 16070.777} C_VEL
LIN {X 0,Y 388.045,Z 504.552,A -85,B 0,C 180,E1 16068.31,E2 16068.31} C_VEL
LIN {X 0,Y 392.545,Z 477.799,A -85,B 0,C 180,E1 16066.487,E2 16066.487} C_VEL
LIN {X 0,Y 394.14,Z 469.642,A -85,B 0,C 180,E1 16065.83,E2 16065.83} C_VEL
LIN {X 0,Y 394.557,Z 466.978,A -85,B 0,C 180,E1 16065.303,E2 16065.303} C_VEL
LIN {X 0,Y 394.266,Z 468.067,A -85,B 0,C 180,E1 16063.614,E2 16063.614} C_VEL
LIN {X 0,Y 394.543,Z 471.186,A -85,B 0,C 180,E1 16062.125,E2 16062.125} C_VEL
LIN {X 0,Y 394.565,Z 471.905,A -85,B 0,C 180,E1 16061.941,E2 16061.941} C_VEL
LIN {X 0,Y 378.873,Z 550.182,A -85,B 0,C 180,E1 16059.183,E2 16059.183} C_VEL
LIN {X 0,Y 368.109,Z 615.728,A -85,B 0,C 180,E1 16056.817,E2 16056.817} C_VEL
LIN {X 0,Y 364.598,Z 640.107,A -85,B 0,C 180,E1 16055.838,E2 16055.838} C_VEL
LIN {X 0,Y 361.148,Z 660.474,A -85,B 0,C 180,E1 16054.706,E2 16054.706} C_VEL
LIN {X 0,Y 357.461,Z 679.296,A -85,B 0,C 180,E1 16053.342,E2 16053.342} C_VEL
LIN {X 0,Y 353.408,Z 697.67,A -85,B 0,C 180,E1 16051.656,E2 16051.656} C_VEL
LIN {X 0,Y 349.281,Z 714.976,A -85,B 0,C 180,E1 16049.685,E2 16049.685} C_VEL
LIN {X 0,Y 345.321,Z 730.521,A -85,B 0,C 180,E1 16047.505,E2 16047.505} C_VEL
LIN {X 0,Y 341.588,Z 744.427,A -85,B 0,C 180,E1 16045.114,E2 16045.114} C_VEL
LIN {X 0,Y 338.091,Z 757.172,A -85,B 0,C 180,E1 16042.426,E2 16042.426} C_VEL
LIN {X 0,Y 335.22,Z 767.668,A -85,B 0,C 180,E1 16039.697,E2 16039.697} C_VEL
LIN {X 0,Y 332.81,Z 776.708,A -85,B 0,C 180,E1 16036.763,E2 16036.763} C_VEL
LIN {X 0,Y 330.925,Z 784.195,A -85,B 0,C 180,E1 16033.631,E2 16033.631} C_VEL
LIN {X 0,Y 329.638,Z 789.71,A -85,B 0,C 180,E1 16030.486,E2 16030.486} C_VEL
LIN {X 0,Y 328.85,Z 793.425,A -85,B 0,C 180,E1 16027.336,E2 16027.336} C_VEL
LIN {X 0,Y 328.43,Z 795.426,A -85,B 0,C 180,E1 16024.19,E2 16024.19} C_VEL
LIN {X 0,Y 328.249,Z 795.733,A -85,B 0,C 180,E1 16021.047,E2 16021.047} C_VEL
LIN {X 0,Y 328.192,Z 794.469,A -85,B 0,C 180,E1 16018.079,E2 16018.079} C_VEL
LIN {X 0,Y 328.251,Z 791.653,A -85,B 0,C 180,E1 16015.107,E2 16015.107} C_VEL
LIN {X 0,Y 328.477,Z 787.211,A -85,B 0,C 180,E1 16012.127,E2 16012.127} C_VEL
LIN {X 0,Y 328.977,Z 780.734,A -85,B 0,C 180,E1 16009.022,E2 16009.022} C_VEL
LIN {X 0,Y 329.789,Z 772.909,A -85,B 0,C 180,E1 16006.142,E2 16006.142} C_VEL
LIN {X 0,Y 331.032,Z 762.954,A -85,B 0,C 180,E1 16003.232,E2 16003.232} C_VEL
LIN {X 0,Y 332.631,Z 751.444,A -85,B 0,C 180,E1 16000.509,E2 16000.509} C_VEL
LIN {X 0,Y 334.487,Z 738.853,A -85,B 0,C 180,E1 15998.059,E2 15998.059} C_VEL
LIN {X 0,Y 336.589,Z 724.709,A -85,B 0,C 180,E1 15995.779,E2 15995.779} C_VEL
LIN {X 0,Y 338.821,Z 709.295,A -85,B 0,C 180,E1 15993.727,E2 15993.727} C_VEL
LIN {X 0,Y 341.016,Z 693,A -85,B 0,C 180,E1 15991.95,E2 15991.95} C_VEL
LIN {X 0,Y 343.156,Z 675.522,A -85,B 0,C 180,E1 15990.404,E2 15990.404} C_VEL
LIN {X 0,Y 345.13,Z 656.836,A -85,B 0,C 180,E1 15989.097,E2 15989.097} C_VEL
LIN {X 0,Y 346.828,Z 636.897,A -85,B 0,C 180,E1 15988.043,E2 15988.043} C_VEL
LIN {X 0,Y 348.138,Z 616.594,A -85,B 0,C 180,E1 15987.293,E2 15987.293} C_VEL
LIN {X 0,Y 357.005,Z 447.889,A -85,B 0,C 180,E1 15982.782,E2 15982.782} C_VEL
LIN {X 0,Y 341.637,Z 415.895,A -85,B 0,C 180,E1 15980.197,E2 15980.197} C_VEL
LIN {X 0,Y 340.387,Z 413.322,A -85,B 0,C 180,E1 15979.962,E2 15979.962} C_VEL
LIN {X 0,Y 333.105,Z 394.083,A -85,B 0,C 180,E1 15976.711,E2 15976.711} C_VEL
LIN {X 0,Y 329.992,Z 385.695,A -85,B 0,C 180,E1 15975.227,E2 15975.227} C_VEL
LIN {X 0,Y 330.004,Z 385.691,A -85,B 0,C 180,E1 15970.878,E2 15970.878} C_VEL
LIN {X 0,Y 330.014,Z 385.692,A -85,B 0,C 180,E1 15966.593,E2 15966.593} C_VEL
LIN {X 0,Y 330.023,Z 385.69,A -85,B 0,C 180,E1 15962.224,E2 15962.224} C_VEL
LIN {X 0,Y 330.017,Z 385.692,A -85,B 0,C 180,E1 15958.009,E2 15958.009} C_VEL
LIN {X 0,Y 330.004,Z 385.688,A -85,B 0,C 180,E1 15953.764,E2 15953.764} C_VEL
LIN {X 0,Y 329.994,Z 385.693,A -85,B 0,C 180,E1 15949.469,E2 15949.469} C_VEL
LIN {X 0,Y 329.985,Z 385.694,A -85,B 0,C 180,E1 15945.105,E2 15945.105} C_VEL
LIN {X 0,Y 329.99,Z 385.693,A -85,B 0,C 180,E1 15940.828,E2 15940.828} C_VEL
LIN {X 0,Y 329.996,Z 385.69,A -85,B 0,C 180,E1 15936.612,E2 15936.612} C_VEL
LIN {X 0,Y 330.009,Z 385.686,A -85,B 0,C 180,E1 15932.257,E2 15932.257} C_VEL
LIN {X 0,Y 330.016,Z 385.681,A -85,B 0,C 180,E1 15928.09,E2 15928.09} C_VEL
LIN {X 0,Y 330.019,Z 385.686,A -85,B 0,C 180,E1 15923.738,E2 15923.738} C_VEL
LIN {X 0,Y 330.008,Z 385.691,A -85,B 0,C 180,E1 15919.526,E2 15919.526} C_VEL
LIN {X 0,Y 329.991,Z 385.694,A -85,B 0,C 180,E1 15915.142,E2 15915.142} C_VEL
LIN {X 0,Y 329.989,Z 385.693,A -85,B 0,C 180,E1 15910.899,E2 15910.899} C_VEL
LIN {X 0,Y 329.986,Z 385.691,A -85,B 0,C 180,E1 15906.613,E2 15906.613} C_VEL
LIN {X 0,Y 329.997,Z 385.69,A -85,B 0,C 180,E1 15902.219,E2 15902.219} C_VEL
LIN {X 0,Y 330.006,Z 385.693,A -85,B 0,C 180,E1 15897.979,E2 15897.979} C_VEL
LIN {X 0,Y 330.014,Z 385.695,A -85,B 0,C 180,E1 15895.486,E2 15895.486} C_VEL
LIN {X 0,Y 329.011,Z 385.822,A -85,B 0,C 180,E1 15894.149,E2 15894.149} C_VEL
LIN {X 0,Y 324.302,Z 386.406,A -85,B 0,C 180,E1 15891.523,E2 15891.523} C_VEL
LIN {X 0,Y 322.192,Z 386.667,A -85,B 0,C 180,E1 15889.772,E2 15889.772} C_VEL
LIN {X 0,Y 322.081,Z 386.682,A -85,B 0,C 180,E1 15889.373,E2 15889.373} C_VEL
LIN {X 0,Y 322.058,Z 386.683,A -85,B 0,C 180,E1 15884.939,E2 15884.939} C_VEL
LIN {X 0,Y 322.092,Z 386.902,A -85,B 0,C 180,E1 15883.025,E2 15883.025} C_VEL
LIN {X 0,Y 326.985,Z 403.591,A -85,B 0,C 180,E1 15879.041,E2 15879.041} C_VEL
LIN {X 0,Y 331.427,Z 419.925,A -85,B 0,C 180,E1 15875.397,E2 15875.397} C_VEL
LIN {X 0,Y 334.551,Z 432.991,A -85,B 0,C 180,E1 15872.647,E2 15872.647} C_VEL
LIN {X 0,Y 331.085,Z 459.153,A -85,B 0,C 180,E1 15868.107,E2 15868.107} C_VEL
LIN {X 0,Y 329.01,Z 477.814,A -85,B 0,C 180,E1 15864.958,E2 15864.958} C_VEL
LIN {X 0,Y 332.885,Z 513.08,A -85,B 0,C 180,E1 15863.499,E2 15863.499} C_VEL
LIN {X 0,Y 328.706,Z 609.616,A -85,B 0,C 180,E1 15860.406,E2 15860.406} C_VEL
LIN {X 0,Y 327.971,Z 626.455,A -85,B 0,C 180,E1 15859.548,E2 15859.548} C_VEL
LIN {X 0,Y 327.002,Z 643.122,A -85,B 0,C 180,E1 15858.357,E2 15858.357} C_VEL
LIN {X 0,Y 325.88,Z 659.038,A -85,B 0,C 180,E1 15856.855,E2 15856.855} C_VEL
LIN {X 0,Y 324.82,Z 673.689,A -85,B 0,C 180,E1 15855.077,E2 15855.077} C_VEL
LIN {X 0,Y 323.779,Z 687.546,A -85,B 0,C 180,E1 15852.938,E2 15852.938} C_VEL
LIN {X 0,Y 322.967,Z 698.937,A -85,B 0,C 180,E1 15850.705,E2 15850.705} C_VEL
LIN {X 0,Y 322.412,Z 708.301,A -85,B 0,C 180,E1 15848.381,E2 15848.381} C_VEL
LIN {X 0,Y 322.096,Z 715.652,A -85,B 0,C 180,E1 15846.059,E2 15846.059} C_VEL
LIN {X 0,Y 322.008,Z 721.856,A -85,B 0,C 180,E1 15843.382,E2 15843.382} C_VEL
LIN {X 0,Y 322.178,Z 725.778,A -85,B 0,C 180,E1 15840.889,E2 15840.889} C_VEL
LIN {X 0,Y 322.602,Z 728.116,A -85,B 0,C 180,E1 15838.224,E2 15838.224} C_VEL
LIN {X 0,Y 323.281,Z 728.545,A -85,B 0,C 180,E1 15835.743,E2 15835.743} C_VEL
LIN {X 0,Y 324.364,Z 727.114,A -85,B 0,C 180,E1 15833.015,E2 15833.015} C_VEL
LIN {X 0,Y 325.774,Z 723.846,A -85,B 0,C 180,E1 15830.46,E2 15830.46} C_VEL
LIN {X 0,Y 327.511,Z 718.947,A -85,B 0,C 180,E1 15828.019,E2 15828.019} C_VEL
LIN {X 0,Y 329.633,Z 712.041,A -85,B 0,C 180,E1 15825.598,E2 15825.598} C_VEL
LIN {X 0,Y 332.011,Z 703.738,A -85,B 0,C 180,E1 15823.376,E2 15823.376} C_VEL
LIN {X 0,Y 334.746,Z 693.114,A -85,B 0,C 180,E1 15821.181,E2 15821.181} C_VEL
LIN {X 0,Y 337.494,Z 681.473,A -85,B 0,C 180,E1 15819.266,E2 15819.266} C_VEL
LIN {X 0,Y 340.625,Z 667.025,A -85,B 0,C 180,E1 15817.385,E2 15817.385} C_VEL
LIN {X 0,Y 343.641,Z 651.172,A -85,B 0,C 180,E1 15815.779,E2 15815.779} C_VEL
LIN {X 0,Y 346.491,Z 634.198,A -85,B 0,C 180,E1 15814.443,E2 15814.443} C_VEL
LIN {X 0,Y 349.081,Z 615.254,A -85,B 0,C 180,E1 15813.357,E2 15813.357} C_VEL
LIN {X 0,Y 363.005,Z 526.336,A -85,B 0,C 180,E1 15809.469,E2 15809.469} C_VEL
LIN {X 0,Y 362.892,Z 510.617,A -85,B 0,C 180,E1 15807.901,E2 15807.901} C_VEL
LIN {X 0,Y 362.654,Z 495.652,A -85,B 0,C 180,E1 15806.087,E2 15806.087} C_VEL
LIN {X 0,Y 362.661,Z 481.354,A -85,B 0,C 180,E1 15803.99,E2 15803.99} C_VEL
LIN {X 0,Y 362.901,Z 475.809,A -85,B 0,C 180,E1 15803.036,E2 15803.036} C_VEL
LIN {X 0,Y 363.683,Z 472.285,A -85,B 0,C 180,E1 15800.778,E2 15800.778} C_VEL
LIN {X 0,Y 364.247,Z 470.824,A -85,B 0,C 180,E1 15799,E2 15799} C_VEL
LIN {X 0,Y 365.234,Z 470.26,A -85,B 0,C 180,E1 15796.736,E2 15796.736} C_VEL
LIN {X 0,Y 365.77,Z 473.172,A -85,B 0,C 180,E1 15793.921,E2 15793.921} C_VEL
LIN {X 0,Y 367.34,Z 476.684,A -85,B 0,C 180,E1 15792.68,E2 15792.68} C_VEL
LIN {X 0,Y 367.157,Z 491.843,A -85,B 0,C 180,E1 15791.283,E2 15791.283} C_VEL
LIN {X 0,Y 366.634,Z 501.654,A -85,B 0,C 180,E1 15790.638,E2 15790.638} C_VEL
LIN {X 0,Y 358.569,Z 562.517,A -85,B 0,C 180,E1 15788.539,E2 15788.539} C_VEL
LIN {X 0,Y 351.303,Z 630.728,A -85,B 0,C 180,E1 15786.306,E2 15786.306} C_VEL
LIN {X 0,Y 348.567,Z 657.534,A -85,B 0,C 180,E1 15785.392,E2 15785.392} C_VEL
LIN {X 0,Y 345.585,Z 676.792,A -85,B 0,C 180,E1 15784.446,E2 15784.446} C_VEL
LIN {X 0,Y 342.157,Z 695.259,A -85,B 0,C 180,E1 15783.225,E2 15783.225} C_VEL
LIN {X 0,Y 338.541,Z 712.76,A -85,B 0,C 180,E1 15781.716,E2 15781.716} C_VEL
LIN {X 0,Y 334.883,Z 729.372,A -85,B 0,C 180,E1 15779.908,E2 15779.908} C_VEL
LIN {X 0,Y 331.188,Z 745.649,A -85,B 0,C 180,E1 15777.706,E2 15777.706} C_VEL
LIN {X 0,Y 327.841,Z 760.809,A -85,B 0,C 180,E1 15775.179,E2 15775.179} C_VEL
LIN {X 0,Y 325.753,Z 771.765,A -85,B 0,C 180,E1 15773.134,E2 15773.134} C_VEL
LIN {X 0,Y 323.826,Z 785.335,A -85,B 0,C 180,E1 15770.609,E2 15770.609} C_VEL
LIN {X 0,Y 322.266,Z 797.334,A -85,B 0,C 180,E1 15767.888,E2 15767.888} C_VEL
LIN {X 0,Y 321.171,Z 807.757,A -85,B 0,C 180,E1 15764.975,E2 15764.975} C_VEL
LIN {X 0,Y 320.53,Z 816.041,A -85,B 0,C 180,E1 15762.064,E2 15762.064} C_VEL
LIN {X 0,Y 320.28,Z 822.803,A -85,B 0,C 180,E1 15758.98,E2 15758.98} C_VEL
LIN {X 0,Y 320.303,Z 827.663,A -85,B 0,C 180,E1 15755.913,E2 15755.913} C_VEL
LIN {X 0,Y 320.385,Z 830.732,A -85,B 0,C 180,E1 15752.862,E2 15752.862} C_VEL
LIN {X 0,Y 320.424,Z 832.05,A -85,B 0,C 180,E1 15750,E2 15750} C_VEL
LIN {X 0,Y 320.311,Z 831.797,A -85,B 0,C 180,E1 15746.958,E2 15746.958} C_VEL
LIN {X 0,Y 320.192,Z 829.901,A -85,B 0,C 180,E1 15743.905,E2 15743.905} C_VEL
LIN {X 0,Y 320.21,Z 826.374,A -85,B 0,C 180,E1 15740.837,E2 15740.837} C_VEL
LIN {X 0,Y 320.591,Z 821.19,A -85,B 0,C 180,E1 15737.756,E2 15737.756} C_VEL
LIN {X 0,Y 321.574,Z 813.818,A -85,B 0,C 180,E1 15734.49,E2 15734.49} C_VEL
LIN {X 0,Y 323.175,Z 804.924,A -85,B 0,C 180,E1 15731.417,E2 15731.417} C_VEL
LIN {X 0,Y 325.539,Z 793.955,A -85,B 0,C 180,E1 15728.373,E2 15728.373} C_VEL
LIN {X 0,Y 328.629,Z 781.065,A -85,B 0,C 180,E1 15725.465,E2 15725.465} C_VEL
LIN {X 0,Y 332.322,Z 766.459,A -85,B 0,C 180,E1 15722.785,E2 15722.785} C_VEL
LIN {X 0,Y 336.526,Z 750.293,A -85,B 0,C 180,E1 15720.35,E2 15720.35} C_VEL
LIN {X 0,Y 340.909,Z 733.426,A -85,B 0,C 180,E1 15718.271,E2 15718.271} C_VEL
LIN {X 0,Y 345.523,Z 715.224,A -85,B 0,C 180,E1 15716.447,E2 15716.447} C_VEL
LIN {X 0,Y 350.253,Z 695.597,A -85,B 0,C 180,E1 15714.885,E2 15714.885} C_VEL
LIN {X 0,Y 354.854,Z 674.97,A -85,B 0,C 180,E1 15713.621,E2 15713.621} C_VEL
LIN {X 0,Y 359.273,Z 652.075,A -85,B 0,C 180,E1 15712.567,E2 15712.567} C_VEL
LIN {X 0,Y 371.704,Z 576.992,A -85,B 0,C 180,E1 15709.784,E2 15709.784} C_VEL
LIN {X 0,Y 385.851,Z 506.595,A -85,B 0,C 180,E1 15707.206,E2 15707.206} C_VEL
LIN {X 0,Y 391.098,Z 480.579,A -85,B 0,C 180,E1 15705.405,E2 15705.405} C_VEL
LIN {X 0,Y 392.421,Z 474.858,A -85,B 0,C 180,E1 15704.953,E2 15704.953} C_VEL
LIN {X 0,Y 392.222,Z 475.809,A -85,B 0,C 180,E1 15703.764,E2 15703.764} C_VEL
LIN {X 0,Y 392.201,Z 477.558,A -85,B 0,C 180,E1 15702.924,E2 15702.924} C_VEL
LIN {X 0,Y 375.17,Z 556.295,A -85,B 0,C 180,E1 15700.131,E2 15700.131} C_VEL
LIN {X 0,Y 363.456,Z 621.746,A -85,B 0,C 180,E1 15697.716,E2 15697.716} C_VEL
LIN {X 0,Y 359.747,Z 644.465,A -85,B 0,C 180,E1 15696.732,E2 15696.732} C_VEL
LIN {X 0,Y 355.937,Z 664.249,A -85,B 0,C 180,E1 15695.555,E2 15695.555} C_VEL
LIN {X 0,Y 351.646,Z 683.504,A -85,B 0,C 180,E1 15694.066,E2 15694.066} C_VEL
LIN {X 0,Y 347.183,Z 701.732,A -85,B 0,C 180,E1 15692.291,E2 15692.291} C_VEL
LIN {X 0,Y 342.802,Z 718.203,A -85,B 0,C 180,E1 15690.304,E2 15690.304} C_VEL
LIN {X 0,Y 338.445,Z 733.616,A -85,B 0,C 180,E1 15688.017,E2 15688.017} C_VEL
LIN {X 0,Y 334.378,Z 747.448,A -85,B 0,C 180,E1 15685.505,E2 15685.505} C_VEL
LIN {X 0,Y 330.67,Z 759.828,A -85,B 0,C 180,E1 15682.743,E2 15682.743} C_VEL
LIN {X 0,Y 327.492,Z 770.366,A -85,B 0,C 180,E1 15679.809,E2 15679.809} C_VEL
LIN {X 0,Y 324.971,Z 778.909,A -85,B 0,C 180,E1 15676.811,E2 15676.811} C_VEL
LIN {X 0,Y 322.987,Z 785.987,A -85,B 0,C 180,E1 15673.58,E2 15673.58} C_VEL
LIN {X 0,Y 321.611,Z 791.321,A -85,B 0,C 180,E1 15670.207,E2 15670.207} C_VEL
LIN {X 0,Y 320.827,Z 794.606,A -85,B 0,C 180,E1 15666.981,E2 15666.981} C_VEL
LIN {X 0,Y 320.418,Z 796.19,A -85,B 0,C 180,E1 15663.757,E2 15663.757} C_VEL
LIN {X 0,Y 320.252,Z 796.123,A -85,B 0,C 180,E1 15660.715,E2 15660.715} C_VEL
LIN {X 0,Y 320.204,Z 794.401,A -85,B 0,C 180,E1 15657.494,E2 15657.494} C_VEL
LIN {X 0,Y 320.288,Z 791.156,A -85,B 0,C 180,E1 15654.446,E2 15654.446} C_VEL
LIN {X 0,Y 320.567,Z 786.26,A -85,B 0,C 180,E1 15651.389,E2 15651.389} C_VEL
LIN {X 0,Y 321.142,Z 779.586,A -85,B 0,C 180,E1 15648.324,E2 15648.324} C_VEL
LIN {X 0,Y 322.044,Z 771.503,A -85,B 0,C 180,E1 15645.434,E2 15645.434} C_VEL
LIN {X 0,Y 323.373,Z 761.437,A -85,B 0,C 180,E1 15642.547,E2 15642.547} C_VEL
LIN {X 0,Y 325.054,Z 749.888,A -85,B 0,C 180,E1 15639.848,E2 15639.848} C_VEL
LIN {X 0,Y 327.117,Z 736.302,A -85,B 0,C 180,E1 15637.253,E2 15637.253} C_VEL
LIN {X 0,Y 329.351,Z 721.615,A -85,B 0,C 180,E1 15634.944,E2 15634.944} C_VEL
LIN {X 0,Y 331.747,Z 705.259,A -85,B 0,C 180,E1 15632.831,E2 15632.831} C_VEL
LIN {X 0,Y 334.126,Z 687.849,A -85,B 0,C 180,E1 15631.002,E2 15631.002} C_VEL
LIN {X 0,Y 336.379,Z 669.378,A -85,B 0,C 180,E1 15629.45,E2 15629.45} C_VEL
LIN {X 0,Y 338.311,Z 650.29,A -85,B 0,C 180,E1 15628.21,E2 15628.21} C_VEL
LIN {X 0,Y 339.946,Z 630.135,A -85,B 0,C 180,E1 15627.242,E2 15627.242} C_VEL
LIN {X 0,Y 341.237,Z 607.423,A -85,B 0,C 180,E1 15626.511,E2 15626.511} C_VEL
LIN {X 0,Y 349.928,Z 450.281,A -85,B 0,C 180,E1 15622.191,E2 15622.191} C_VEL
LIN {X 0,Y 335.415,Z 419.924,A -85,B 0,C 180,E1 15619.675,E2 15619.675} C_VEL
LIN {X 0,Y 332.231,Z 413.436,A -85,B 0,C 180,E1 15619.06,E2 15619.06} C_VEL
LIN {X 0,Y 324.666,Z 393.482,A -85,B 0,C 180,E1 15615.601,E2 15615.601} C_VEL
LIN {X 0,Y 322.083,Z 386.678,A -85,B 0,C 180,E1 15614.383,E2 15614.383} C_VEL
LIN {X 0,Y 322.067,Z 386.679,A -85,B 0,C 180,E1 15609.989,E2 15609.989} C_VEL
LIN {X 0,Y 322.057,Z 386.683,A -85,B 0,C 180,E1 15605.709,E2 15605.709} C_VEL
LIN {X 0,Y 322.051,Z 386.682,A -85,B 0,C 180,E1 15601.23,E2 15601.23} C_VEL
LIN {X 0,Y 322.055,Z 386.68,A -85,B 0,C 180,E1 15596.954,E2 15596.954} C_VEL
LIN {X 0,Y 322.065,Z 386.679,A -85,B 0,C 180,E1 15592.641,E2 15592.641} C_VEL
LIN {X 0,Y 322.083,Z 386.678,A -85,B 0,C 180,E1 15588.206,E2 15588.206} C_VEL
LIN {X 0,Y 322.074,Z 386.675,A -85,B 0,C 180,E1 15583.83,E2 15583.83} C_VEL
LIN {X 0,Y 322.055,Z 386.676,A -85,B 0,C 180,E1 15579.471,E2 15579.471} C_VEL
LIN {X 0,Y 322.047,Z 386.678,A -85,B 0,C 180,E1 15575.166,E2 15575.166} C_VEL
LIN {X 0,Y 322.049,Z 386.68,A -85,B 0,C 180,E1 15570.712,E2 15570.712} C_VEL
LIN {X 0,Y 322.057,Z 386.675,A -85,B 0,C 180,E1 15566.44,E2 15566.44} C_VEL
LIN {X 0,Y 322.071,Z 386.672,A -85,B 0,C 180,E1 15562.149,E2 15562.149} C_VEL
LIN {X 0,Y 322.078,Z 386.675,A -85,B 0,C 180,E1 15557.813,E2 15557.813} C_VEL
LIN {X 0,Y 322.076,Z 386.677,A -85,B 0,C 180,E1 15553.59,E2 15553.59} C_VEL
LIN {X 0,Y 322.06,Z 386.679,A -85,B 0,C 180,E1 15549.273,E2 15549.273} C_VEL
LIN {X 0,Y 322.053,Z 386.681,A -85,B 0,C 180,E1 15545.024,E2 15545.024} C_VEL
LIN {X 0,Y 322.048,Z 386.679,A -85,B 0,C 180,E1 15540.624,E2 15540.624} C_VEL
LIN {X 0,Y 322.053,Z 386.686,A -85,B 0,C 180,E1 15536.239,E2 15536.239} C_VEL
LIN {X 0,Y 322.071,Z 386.683,A -85,B 0,C 180,E1 15531.845,E2 15531.845} C_VEL
LIN {X 0,Y 322.081,Z 386.682,A -85,B 0,C 180,E1 15529.373,E2 15529.373} C_VEL
LIN {X 0,Y 321.056,Z 386.811,A -85,B 0,C 180,E1 15528.464,E2 15528.464} C_VEL
LIN {X 0,Y 314.697,Z 387.599,A -85,B 0,C 180,E1 15525.976,E2 15525.976} C_VEL
LIN {X 0,Y 314.134,Z 387.669,A -85,B 0,C 180,E1 15525.297,E2 15525.297} C_VEL
LIN {X 0,Y 314.156,Z 387.875,A -85,B 0,C 180,E1 15523.804,E2 15523.804} C_VEL
LIN {X 0,Y 318.943,Z 404.11,A -85,B 0,C 180,E1 15519.82,E2 15519.82} C_VEL
LIN {X 0,Y 323.541,Z 421.062,A -85,B 0,C 180,E1 15515.935,E2 15515.935} C_VEL
LIN {X 0,Y 326.921,Z 434.971,A -85,B 0,C 180,E1 15512.932,E2 15512.932} C_VEL
LIN {X 0,Y 323.274,Z 461.498,A -85,B 0,C 180,E1 15508.244,E2 15508.244} C_VEL
LIN {X 0,Y 321.394,Z 477.657,A -85,B 0,C 180,E1 15505.465,E2 15505.465} C_VEL
LIN {X 0,Y 325.279,Z 513.923,A -85,B 0,C 180,E1 15503.926,E2 15503.926} C_VEL
LIN {X 0,Y 320.944,Z 609.601,A -85,B 0,C 180,E1 15500.749,E2 15500.749} C_VEL
LIN {X 0,Y 320.168,Z 626.807,A -85,B 0,C 180,E1 15499.854,E2 15499.854} C_VEL
LIN {X 0,Y 319.168,Z 643.579,A -85,B 0,C 180,E1 15498.635,E2 15498.635} C_VEL
LIN {X 0,Y 318.013,Z 659.6,A -85,B 0,C 180,E1 15497.097,E2 15497.097} C_VEL
LIN {X 0,Y 316.919,Z 674.368,A -85,B 0,C 180,E1 15495.274,E2 15495.274} C_VEL
LIN {X 0,Y 315.848,Z 688.348,A -85,B 0,C 180,E1 15493.082,E2 15493.082} C_VEL
LIN {X 0,Y 315.018,Z 699.851,A -85,B 0,C 180,E1 15490.793,E2 15490.793} C_VEL
LIN {X 0,Y 314.484,Z 708.662,A -85,B 0,C 180,E1 15488.587,E2 15488.587} C_VEL
LIN {X 0,Y 314.133,Z 716.69,A -85,B 0,C 180,E1 15486.029,E2 15486.029} C_VEL
LIN {X 0,Y 314.058,Z 722.633,A -85,B 0,C 180,E1 15483.468,E2 15483.468} C_VEL
LIN {X 0,Y 314.246,Z 726.815,A -85,B 0,C 180,E1 15480.912,E2 15480.912} C_VEL
LIN {X 0,Y 314.699,Z 729.328,A -85,B 0,C 180,E1 15478.18,E2 15478.18} C_VEL
LIN {X 0,Y 315.439,Z 730.019,A -85,B 0,C 180,E1 15475.637,E2 15475.637} C_VEL
LIN {X 0,Y 316.56,Z 728.853,A -85,B 0,C 180,E1 15472.924,E2 15472.924} C_VEL
LIN {X 0,Y 318.136,Z 725.846,A -85,B 0,C 180,E1 15470.229,E2 15470.229} C_VEL
LIN {X 0,Y 320.136,Z 720.758,A -85,B 0,C 180,E1 15467.555,E2 15467.555} C_VEL
LIN {X 0,Y 322.286,Z 714.666,A -85,B 0,C 180,E1 15465.262,E2 15465.262} C_VEL
LIN {X 0,Y 325.234,Z 705.286,A -85,B 0,C 180,E1 15462.65,E2 15462.65} C_VEL
LIN {X 0,Y 328.211,Z 694.792,A -85,B 0,C 180,E1 15460.421,E2 15460.421} C_VEL
LIN {X 0,Y 331.341,Z 682.833,A -85,B 0,C 180,E1 15458.399,E2 15458.399} C_VEL
LIN {X 0,Y 334.737,Z 668.498,A -85,B 0,C 180,E1 15456.493,E2 15456.493} C_VEL
LIN {X 0,Y 338.01,Z 653.121,A -85,B 0,C 180,E1 15454.882,E2 15454.882} C_VEL
LIN {X 0,Y 341.249,Z 635.517,A -85,B 0,C 180,E1 15453.46,E2 15453.46} C_VEL
LIN {X 0,Y 344.062,Z 616.98,A -85,B 0,C 180,E1 15452.363,E2 15452.363} C_VEL
LIN {X 0,Y 358.914,Z 528.599,A -85,B 0,C 180,E1 15448.418,E2 15448.418} C_VEL
LIN {X 0,Y 359.208,Z 513.253,A -85,B 0,C 180,E1 15446.818,E2 15446.818} C_VEL
LIN {X 0,Y 359.462,Z 498.588,A -85,B 0,C 180,E1 15444.943,E2 15444.943} C_VEL
LIN {X 0,Y 360.006,Z 486.093,A -85,B 0,C 180,E1 15443.038,E2 15443.038} C_VEL
LIN {X 0,Y 360.256,Z 482.387,A -85,B 0,C 180,E1 15442.368,E2 15442.368} C_VEL
LIN {X 0,Y 359.767,Z 478.723,A -85,B 0,C 180,E1 15440.267,E2 15440.267} C_VEL
LIN {X 0,Y 359.98,Z 477.41,A -85,B 0,C 180,E1 15438.62,E2 15438.62} C_VEL
LIN {X 0,Y 361.021,Z 477.084,A -85,B 0,C 180,E1 15436.752,E2 15436.752} C_VEL
LIN {X 0,Y 363.264,Z 480.494,A -85,B 0,C 180,E1 15434.243,E2 15434.243} C_VEL
LIN {X 0,Y 364.206,Z 482.688,A -85,B 0,C 180,E1 15433.449,E2 15433.449} C_VEL
LIN {X 0,Y 363.568,Z 496.667,A -85,B 0,C 180,E1 15432.162,E2 15432.162} C_VEL
LIN {X 0,Y 362.659,Z 506.12,A -85,B 0,C 180,E1 15431.6,E2 15431.6} C_VEL
LIN {X 0,Y 352.17,Z 578.778,A -85,B 0,C 180,E1 15429.072,E2 15429.072} C_VEL
LIN {X 0,Y 343.385,Z 655.644,A -85,B 0,C 180,E1 15426.448,E2 15426.448} C_VEL
LIN {X 0,Y 340.406,Z 673.8,A -85,B 0,C 180,E1 15425.562,E2 15425.562} C_VEL
LIN {X 0,Y 336.491,Z 693.35,A -85,B 0,C 180,E1 15424.27,E2 15424.27} C_VEL
LIN {X 0,Y 332.409,Z 711.605,A -85,B 0,C 180,E1 15422.679,E2 15422.679} C_VEL
LIN {X 0,Y 328.495,Z 727.912,A -85,B 0,C 180,E1 15420.869,E2 15420.869} C_VEL
LIN {X 0,Y 324.48,Z 744.159,A -85,B 0,C 180,E1 15418.631,E2 15418.631} C_VEL
LIN {X 0,Y 320.824,Z 759.243,A -85,B 0,C 180,E1 15416.068,E2 15416.068} C_VEL
LIN {X 0,Y 317.853,Z 772.293,A -85,B 0,C 180,E1 15413.351,E2 15413.351} C_VEL
LIN {X 0,Y 315.404,Z 788.737,A -85,B 0,C 180,E1 15410.021,E2 15410.021} C_VEL
